   LaserStart_Ext()
   LIN {X -4.398, Y -8.592, Z 58.650}
   LaserEnd_Ext()
   LIN {X -4.398, Y 35.301, Z 58.650}
   LaserStart_Ext()
   LIN {X -4.398, Y 43.362, Z 58.650}
   LaserEnd_Ext()
   LIN {X -5.398, Y 42.761, Z 58.650}
   LaserStart_Ext()
   LIN {X -5.398, Y 38.302, Z 58.650}
   LaserEnd_Ext()
   LIN {X -5.398, Y -11.620, Z 58.650}
   LaserStart_Ext()
   LIN {X -5.398, Y -17.297, Z 58.650}
   LaserEnd_Ext()
   LIN {X -5.398, Y -23.853, Z 58.650}
   LaserStart_Ext()
   LIN {X -5.398, Y -26.825, Z 58.650}
   LaserEnd_Ext()
   LIN {X -6.398, Y -25.920, Z 58.650}
   LaserStart_Ext()
   LIN {X -6.398, Y -20.860, Z 58.650}
   LaserEnd_Ext()
   LIN {X -6.398, Y -20.280, Z 58.650}
   LaserStart_Ext()
   LIN {X -6.398, Y -14.254, Z 58.650}
   LaserEnd_Ext()
   LIN {X -7.398, Y -16.609, Z 58.650}
   LaserStart_Ext()
   LIN {X -7.398, Y -24.292, Z 58.650}
   LaserEnd_Ext()
   LIN {X -8.398, Y -20.132, Z 58.650}
   LaserStart_Ext()
   LIN {X -8.398, Y -20.032, Z 58.650}
   LaserEnd_Ext()
   LIN {X 3.651, Y -23.553, Z 59.500}
   LaserStart_Ext()
   LIN {X 2.587, Y -24.503, Z 59.500} C_DIS
   LIN {X 2.113, Y -24.924, Z 59.500} C_DIS
   LIN {X 1.058, Y -25.251, Z 59.500} C_DIS
   LIN {X 0.034, Y -25.570, Z 59.500} C_DIS
   LIN {X -0.602, Y -25.496, Z 59.500} C_DIS
   LIN {X -1.998, Y -25.328, Z 59.500} C_DIS
   LIN {X -3.608, Y -24.363, Z 59.500} C_DIS
   LIN {X -3.770, Y -24.267, Z 59.500} C_DIS
   LIN {X -3.863, Y -24.136, Z 59.500} C_DIS
   LIN {X -4.971, Y -22.565, Z 59.500} C_DIS
   LIN {X -5.320, Y -20.722, Z 59.500} C_DIS
   LIN {X -5.360, Y -20.515, Z 59.500} C_DIS
   LIN {X -4.561, Y -18.080, Z 59.500} C_DIS
   LIN {X -4.452, Y -17.736, Z 59.500} C_DIS
   LIN {X -3.971, Y -17.280, Z 59.500} C_DIS
   LIN {X -2.945, Y -16.315, Z 59.500} C_DIS
   LIN {X -1.929, Y -15.973, Z 59.500} C_DIS
   LIN {X -0.833, Y -15.606, Z 59.500} C_DIS
   LIN {X 0.602, Y -15.764, Z 59.500} C_DIS
   LIN {X 1.276, Y -15.837, Z 59.500} C_DIS
   LIN {X 1.727, Y -16.111, Z 59.500} C_DIS
   LIN {X 3.095, Y -16.936, Z 59.500} C_DIS
   LIN {X 4.204, Y -18.721, Z 59.500} C_DIS
   LIN {X 4.436, Y -19.097, Z 59.500} C_DIS
   LIN {X 4.464, Y -19.505, Z 59.500} C_DIS
   LIN {X 4.594, Y -21.301, Z 59.500} C_DIS
   LIN {X 4.218, Y -22.204, Z 59.500} C_DIS
   LIN {X 3.651, Y -23.553, Z 59.500}
   LaserEnd_Ext()
   LIN {X 4.394, Y 32.266, Z 59.500}
   LaserStart_Ext()
   LIN {X 4.205, Y 32.926, Z 59.500} C_DIS
   LIN {X 4.104, Y 33.232, Z 59.500} C_DIS
   LIN {X 3.655, Y 34.459, Z 59.500} C_DIS
   LIN {X 2.800, Y 36.803, Z 59.500} C_DIS
   LIN {X 2.432, Y 37.727, Z 59.500} C_DIS
   LIN {X 1.920, Y 39.018, Z 59.500} C_DIS
   LIN {X 1.377, Y 40.311, Z 59.500} C_DIS
   LIN {X 1.096, Y 40.976, Z 59.500} C_DIS
   LIN {X 0.783, Y 41.682, Z 59.500} C_DIS
   LIN {X 0.407, Y 42.537, Z 59.500} C_DIS
   LIN {X 0.002, Y 43.122, Z 59.500} C_DIS
   LIN {X -0.432, Y 43.746, Z 59.500} C_DIS
   LIN {X -1.529, Y 44.437, Z 59.500} C_DIS
   LIN {X -1.904, Y 44.674, Z 59.500} C_DIS
   LIN {X -2.162, Y 44.707, Z 59.500} C_DIS
   LIN {X -3.636, Y 44.890, Z 59.500} C_DIS
   LIN {X -5.139, Y 44.206, Z 59.500} C_DIS
   LIN {X -5.994, Y 43.806, Z 59.500} C_DIS
   LIN {X -6.906, Y 42.487, Z 59.500} C_DIS
   LIN {X -7.065, Y 41.690, Z 59.500} C_DIS
   LIN {X -7.219, Y 40.882, Z 59.500} C_DIS
   LIN {X -7.097, Y 40.290, Z 59.500} C_DIS
   LIN {X -6.944, Y 39.491, Z 59.500} C_DIS
   LIN {X -6.557, Y 38.443, Z 59.500} C_DIS
   LIN {X -6.510, Y 38.317, Z 59.500} C_DIS
   LIN {X -6.469, Y 38.202, Z 59.500} C_DIS
   LIN {X -5.976, Y 36.809, Z 59.500} C_DIS
   LIN {X -5.262, Y 34.603, Z 59.500} C_DIS
   LIN {X -5.221, Y 34.465, Z 59.500} C_DIS
   LIN {X -4.434, Y 31.691, Z 59.500} C_DIS
   LIN {X -4.225, Y 30.834, Z 59.500} C_DIS
   LIN {X -3.738, Y 28.801, Z 59.500} C_DIS
   LIN {X -2.893, Y 24.053, Z 59.500} C_DIS
   LIN {X -2.741, Y 23.217, Z 59.500} C_DIS
   LIN {X -2.690, Y 22.404, Z 59.500} C_DIS
   LIN {X -2.050, Y 13.702, Z 59.500} C_DIS
   LIN {X -2.396, Y 6.398, Z 59.500} C_DIS
   LIN {X -2.420, Y 5.803, Z 59.500} C_DIS
   LIN {X -2.492, Y 5.299, Z 59.500} C_DIS
   LIN {X -3.366, Y -0.609, Z 59.500} C_DIS
   LIN {X -4.427, Y -5.060, Z 59.500} C_DIS
   LIN {X -4.887, Y -6.944, Z 59.500} C_DIS
   LIN {X -5.301, Y -8.237, Z 59.500} C_DIS
   LIN {X -6.048, Y -10.610, Z 59.500} C_DIS
   LIN {X -6.839, Y -12.728, Z 59.500} C_DIS
   LIN {X -7.391, Y -14.184, Z 59.500} C_DIS
   LIN {X -8.023, Y -15.645, Z 59.500} C_DIS
   LIN {X -8.560, Y -16.902, Z 59.500} C_DIS
   LIN {X -8.871, Y -18.130, Z 59.500} C_DIS
   LIN {X -9.347, Y -19.974, Z 59.500} C_DIS
   LIN {X -9.023, Y -22.429, Z 59.500} C_DIS
   LIN {X -8.856, Y -23.652, Z 59.500} C_DIS
   LIN {X -7.892, Y -25.211, Z 59.500} C_DIS
   LIN {X -6.889, Y -26.844, Z 59.500} C_DIS
   LIN {X -6.353, Y -27.250, Z 59.500} C_DIS
   LIN {X -4.562, Y -28.587, Z 59.500} C_DIS
   LIN {X -4.173, Y -28.761, Z 59.500} C_DIS
   LIN {X -2.604, Y -28.918, Z 59.500} C_DIS
   LIN {X 1.615, Y -29.361, Z 59.500} C_DIS
   LIN {X 2.525, Y -28.992, Z 59.500} C_DIS
   LIN {X 4.880, Y -27.881, Z 59.500} C_DIS
   LIN {X 7.304, Y -25.155, Z 59.500} C_DIS
   LIN {X 7.543, Y -24.875, Z 59.500} C_DIS
   LIN {X 7.671, Y -24.507, Z 59.500} C_DIS
   LIN {X 8.526, Y -22.093, Z 59.500} C_DIS
   LIN {X 8.845, Y -20.129, Z 59.500} C_DIS
   LIN {X 9.042, Y -18.870, Z 59.500} C_DIS
   LIN {X 9.234, Y -17.389, Z 59.500} C_DIS
   LIN {X 9.431, Y -15.935, Z 59.500} C_DIS
   LIN {X 9.570, Y -14.614, Z 59.500} C_DIS
   LIN {X 9.814, Y -12.148, Z 59.500} C_DIS
   LIN {X 10.027, Y -8.821, Z 59.500} C_DIS
   LIN {X 10.110, Y -7.369, Z 59.500} C_DIS
   LIN {X 10.159, Y -2.463, Z 59.500} C_DIS
   LIN {X 10.180, Y -0.855, Z 59.500} C_DIS
   LIN {X 10.169, Y -0.533, Z 59.500} C_DIS
   LIN {X 10.095, Y 1.746, Z 59.500} C_DIS
   LIN {X 9.904, Y 5.040, Z 59.500} C_DIS
   LIN {X 9.462, Y 9.698, Z 59.500} C_DIS
   LIN {X 8.824, Y 13.940, Z 59.500} C_DIS
   LIN {X 7.121, Y 22.903, Z 59.500} C_DIS
   LIN {X 6.371, Y 25.828, Z 59.500} C_DIS
   LIN {X 4.394, Y 32.266, Z 59.500}
   LaserEnd_Ext()
   LIN {X -4.229, Y 43.522, Z 59.500}
   LaserStart_Ext()
   LIN {X -1.952, Y 43.522, Z 59.500}
   LaserEnd_Ext()
   LIN {X -0.798, Y 42.522, Z 59.500}
   LaserStart_Ext()
   LIN {X -5.666, Y 42.522, Z 59.500}
   LaserEnd_Ext()
   LIN {X -6.079, Y 41.522, Z 59.500}
   LaserStart_Ext()
   LIN {X -0.239, Y 41.522, Z 59.500}
   LaserEnd_Ext()
   LIN {X 0.202, Y 40.522, Z 59.500}
   LaserStart_Ext()
   LIN {X -6.124, Y 40.522, Z 59.500}
   LaserEnd_Ext()
   LIN {X -5.889, Y 39.522, Z 59.500}
   LaserStart_Ext()
   LIN {X 0.624, Y 39.522, Z 59.500}
   LaserEnd_Ext()
   LIN {X 1.041, Y 38.522, Z 59.500}
   LaserStart_Ext()
   LIN {X -5.522, Y 38.522, Z 59.500}
   LaserEnd_Ext()
   LIN {X -5.168, Y 37.522, Z 59.500}
   LaserStart_Ext()
   LIN {X 1.438, Y 37.522, Z 59.500}
   LaserEnd_Ext()
   LIN {X 1.835, Y 36.522, Z 59.500}
   LaserStart_Ext()
   LIN {X -4.832, Y 36.522, Z 59.500}
   LaserEnd_Ext()
   LIN {X -4.509, Y 35.522, Z 59.500}
   LaserStart_Ext()
   LIN {X 2.203, Y 35.522, Z 59.500}
   LaserEnd_Ext()
   LIN {X 2.568, Y 34.522, Z 59.500}
   LaserStart_Ext()
   LIN {X -4.198, Y 34.522, Z 59.500}
   LaserEnd_Ext()
   LIN {X -3.914, Y 33.522, Z 59.500}
   LaserStart_Ext()
   LIN {X 2.933, Y 33.522, Z 59.500}
   LaserEnd_Ext()
   LIN {X 3.281, Y 32.522, Z 59.500}
   LaserStart_Ext()
   LIN {X -3.630, Y 32.522, Z 59.500}
   LaserEnd_Ext()
   LIN {X -3.363, Y 31.522, Z 59.500}
   LaserStart_Ext()
   LIN {X 3.576, Y 31.522, Z 59.500}
   LaserEnd_Ext()
   LIN {X 3.883, Y 30.522, Z 59.500}
   LaserStart_Ext()
   LIN {X -3.122, Y 30.522, Z 59.500}
   LaserEnd_Ext()
   LIN {X -2.882, Y 29.522, Z 59.500}
   LaserStart_Ext()
   LIN {X 4.190, Y 29.522, Z 59.500}
   LaserEnd_Ext()
   LIN {X 4.498, Y 28.522, Z 59.500}
   LaserStart_Ext()
   LIN {X -2.672, Y 28.522, Z 59.500}
   LaserEnd_Ext()
   LIN {X -2.494, Y 27.522, Z 59.500}
   LaserStart_Ext()
   LIN {X 4.805, Y 27.522, Z 59.500}
   LaserEnd_Ext()
   LIN {X 5.112, Y 26.522, Z 59.500}
   LaserStart_Ext()
   LIN {X -2.316, Y 26.522, Z 59.500}
   LaserEnd_Ext()
   LIN {X -2.138, Y 25.522, Z 59.500}
   LaserStart_Ext()
   LIN {X 5.417, Y 25.522, Z 59.500}
   LaserEnd_Ext()
   LIN {X 5.673, Y 24.522, Z 59.500}
   LaserStart_Ext()
   LIN {X -1.960, Y 24.522, Z 59.500}
   LaserEnd_Ext()
   LIN {X -1.780, Y 23.522, Z 59.500}
   LaserStart_Ext()
   LIN {X 5.930, Y 23.522, Z 59.500}
   LaserEnd_Ext()
   LIN {X 6.175, Y 22.522, Z 59.500}
   LaserStart_Ext()
   LIN {X -1.695, Y 22.522, Z 59.500}
   LaserEnd_Ext()
   LIN {X -1.622, Y 21.522, Z 59.500}
   LaserStart_Ext()
   LIN {X 6.365, Y 21.522, Z 59.500}
   LaserEnd_Ext()
   LIN {X 6.555, Y 20.522, Z 59.500}
   LaserStart_Ext()
   LIN {X -1.549, Y 20.522, Z 59.500}
   LaserEnd_Ext()
   LIN {X -1.475, Y 19.522, Z 59.500}
   LaserStart_Ext()
   LIN {X 6.745, Y 19.522, Z 59.500}
   LaserEnd_Ext()
   LIN {X 6.936, Y 18.522, Z 59.500}
   LaserStart_Ext()
   LIN {X -1.401, Y 18.522, Z 59.500}
   LaserEnd_Ext()
   LIN {X -1.328, Y 17.522, Z 59.500}
   LaserStart_Ext()
   LIN {X 7.126, Y 17.522, Z 59.500}
   LaserEnd_Ext()
   LIN {X 7.316, Y 16.522, Z 59.500}
   LaserStart_Ext()
   LIN {X -1.254, Y 16.522, Z 59.500}
   LaserEnd_Ext()
   LIN {X -1.181, Y 15.522, Z 59.500}
   LaserStart_Ext()
   LIN {X 7.506, Y 15.522, Z 59.500}
   LaserEnd_Ext()
   LIN {X 7.696, Y 14.522, Z 59.500}
   LaserStart_Ext()
   LIN {X -1.107, Y 14.522, Z 59.500}
   LaserEnd_Ext()
   LIN {X -1.057, Y 13.522, Z 59.500}
   LaserStart_Ext()
   LIN {X 7.876, Y 13.522, Z 59.500}
   LaserEnd_Ext()
   LIN {X 8.027, Y 12.522, Z 59.500}
   LaserStart_Ext()
   LIN {X -1.105, Y 12.522, Z 59.500}
   LaserEnd_Ext()
   LIN {X -1.152, Y 11.522, Z 59.500}
   LaserStart_Ext()
   LIN {X 8.177, Y 11.522, Z 59.500}
   LaserEnd_Ext()
   LIN {X 8.327, Y 10.522, Z 59.500}
   LaserStart_Ext()
   LIN {X -1.199, Y 10.522, Z 59.500}
   LaserEnd_Ext()
   LIN {X -1.247, Y 9.522, Z 59.500}
   LaserStart_Ext()
   LIN {X 8.475, Y 9.522, Z 59.500}
   LaserEnd_Ext()
   LIN {X 8.569, Y 8.522, Z 59.500}
   LaserStart_Ext()
   LIN {X -1.294, Y 8.522, Z 59.500}
   LaserEnd_Ext()
   LIN {X -1.341, Y 7.522, Z 59.500}
   LaserStart_Ext()
   LIN {X 8.664, Y 7.522, Z 59.500}
   LaserEnd_Ext()
   LIN {X 8.759, Y 6.522, Z 59.500}
   LaserStart_Ext()
   LIN {X -1.389, Y 6.522, Z 59.500}
   LaserEnd_Ext()
   LIN {X -1.450, Y 5.522, Z 59.500}
   LaserStart_Ext()
   LIN {X 8.853, Y 5.522, Z 59.500}
   LaserEnd_Ext()
   LIN {X 8.932, Y 4.522, Z 59.500}
   LaserStart_Ext()
   LIN {X -1.596, Y 4.522, Z 59.500}
   LaserEnd_Ext()
   LIN {X -1.744, Y 3.522, Z 59.500}
   LaserStart_Ext()
   LIN {X 8.990, Y 3.522, Z 59.500}
   LaserEnd_Ext()
   LIN {X 9.049, Y 2.522, Z 59.500}
   LaserStart_Ext()
   LIN {X -1.892, Y 2.522, Z 59.500}
   LaserEnd_Ext()
   LIN {X -2.040, Y 1.522, Z 59.500}
   LaserStart_Ext()
   LIN {X 9.102, Y 1.522, Z 59.500}
   LaserEnd_Ext()
   LIN {X 9.135, Y 0.522, Z 59.500}
   LaserStart_Ext()
   LIN {X -2.188, Y 0.522, Z 59.500}
   LaserEnd_Ext()
   LIN {X -2.336, Y -0.478, Z 59.500}
   LaserStart_Ext()
   LIN {X 9.167, Y -0.478, Z 59.500}
   LaserEnd_Ext()
   LIN {X 9.172, Y -1.478, Z 59.500}
   LaserStart_Ext()
   LIN {X -2.545, Y -1.478, Z 59.500}
   LaserEnd_Ext()
   LIN {X -2.784, Y -2.478, Z 59.500}
   LaserStart_Ext()
   LIN {X 9.159, Y -2.478, Z 59.500}
   LaserEnd_Ext()
   LIN {X 9.149, Y -3.478, Z 59.500}
   LaserStart_Ext()
   LIN {X -3.022, Y -3.478, Z 59.500}
   LaserEnd_Ext()
   LIN {X -3.260, Y -4.478, Z 59.500}
   LaserStart_Ext()
   LIN {X 9.139, Y -4.478, Z 59.500}
   LaserEnd_Ext()
   LIN {X 9.129, Y -5.478, Z 59.500}
   LaserStart_Ext()
   LIN {X -3.500, Y -5.478, Z 59.500}
   LaserEnd_Ext()
   LIN {X -3.744, Y -6.478, Z 59.500}
   LaserStart_Ext()
   LIN {X 9.119, Y -6.478, Z 59.500}
   LaserEnd_Ext()
   LIN {X 9.102, Y -7.478, Z 59.500}
   LaserStart_Ext()
   LIN {X -4.008, Y -7.478, Z 59.500}
   LaserEnd_Ext()
   LIN {X -4.329, Y -8.478, Z 59.500}
   LaserStart_Ext()
   LIN {X 9.045, Y -8.478, Z 59.500}
   LaserEnd_Ext()
   LIN {X 8.983, Y -9.478, Z 59.500}
   LaserStart_Ext()
   LIN {X -4.644, Y -9.478, Z 59.500}
   LaserEnd_Ext()
   LIN {X -4.958, Y -10.478, Z 59.500}
   LaserStart_Ext()
   LIN {X 8.919, Y -10.478, Z 59.500}
   LaserEnd_Ext()
   LIN {X 8.855, Y -11.478, Z 59.500}
   LaserStart_Ext()
   LIN {X -5.305, Y -11.478, Z 59.500}
   LaserEnd_Ext()
   LIN {X -5.678, Y -12.478, Z 59.500}
   LaserStart_Ext()
   LIN {X 8.776, Y -12.478, Z 59.500}
   LaserEnd_Ext()
   LIN {X 8.677, Y -13.478, Z 59.500}
   LaserStart_Ext()
   LIN {X -6.054, Y -13.478, Z 59.500}
   LaserEnd_Ext()
   LIN {X -6.434, Y -14.478, Z 59.500}
   LaserStart_Ext()
   LIN {X 8.579, Y -14.478, Z 59.500}
   LaserEnd_Ext()
   LIN {X 8.473, Y -15.478, Z 59.500}
   LaserStart_Ext()
   LIN {X 2.614, Y -15.478, Z 59.500}
   LaserEnd_Ext()
   LIN {X -3.490, Y -15.478, Z 59.500}
   LaserStart_Ext()
   LIN {X -6.862, Y -15.478, Z 59.500}
   LaserEnd_Ext()
   LIN {X -7.292, Y -16.478, Z 59.500}
   LaserStart_Ext()
   LIN {X -4.578, Y -16.478, Z 59.500}
   LaserEnd_Ext()
   LIN {X 3.988, Y -16.478, Z 59.500}
   LaserStart_Ext()
   LIN {X 8.348, Y -16.478, Z 59.500}
   LaserEnd_Ext()
   LIN {X 8.214, Y -17.478, Z 59.500}
   LaserStart_Ext()
   LIN {X 4.609, Y -17.478, Z 59.500}
   LaserEnd_Ext()
   LIN {X -5.419, Y -17.478, Z 59.500}
   LaserStart_Ext()
   LIN {X -7.675, Y -17.478, Z 59.500}
   LaserEnd_Ext()
   LIN {X -7.928, Y -18.478, Z 59.500}
   LaserStart_Ext()
   LIN {X -5.744, Y -18.478, Z 59.500}
   LaserEnd_Ext()
   LIN {X 5.229, Y -18.478, Z 59.500}
   LaserStart_Ext()
   LIN {X 8.085, Y -18.478, Z 59.500}
   LaserEnd_Ext()
   LIN {X 7.935, Y -19.478, Z 59.500}
   LaserStart_Ext()
   LIN {X 5.464, Y -19.478, Z 59.500}
   LaserEnd_Ext()
   LIN {X -6.072, Y -19.478, Z 59.500}
   LaserStart_Ext()
   LIN {X -8.186, Y -19.478, Z 59.500}
   LaserEnd_Ext()
   LIN {X -8.272, Y -20.478, Z 59.500}
   LaserStart_Ext()
   LIN {X -6.358, Y -20.478, Z 59.500}
   LaserEnd_Ext()
   LIN {X 5.537, Y -20.478, Z 59.500}
   LaserStart_Ext()
   LIN {X 7.775, Y -20.478, Z 59.500}
   LaserEnd_Ext()
   LIN {X 7.612, Y -21.478, Z 59.500}
   LaserStart_Ext()
   LIN {X 5.577, Y -21.478, Z 59.500}
   LaserEnd_Ext()
   LIN {X -6.194, Y -21.478, Z 59.500}
   LaserStart_Ext()
   LIN {X -8.140, Y -21.478, Z 59.500}
   LaserEnd_Ext()
   LIN {X -8.007, Y -22.478, Z 59.500}
   LaserStart_Ext()
   LIN {X -6.005, Y -22.478, Z 59.500}
   LaserEnd_Ext()
   LIN {X 5.187, Y -22.478, Z 59.500}
   LaserStart_Ext()
   LIN {X 7.328, Y -22.478, Z 59.500}
   LaserEnd_Ext()
   LIN {X 6.974, Y -23.478, Z 59.500}
   LaserStart_Ext()
   LIN {X 4.768, Y -23.478, Z 59.500}
   LaserEnd_Ext()
   LIN {X -5.550, Y -23.478, Z 59.500}
   LaserStart_Ext()
   LIN {X -7.787, Y -23.478, Z 59.500}
   LaserEnd_Ext()
   LIN {X -7.169, Y -24.478, Z 59.500}
   LaserStart_Ext()
   LIN {X -4.845, Y -24.478, Z 59.500}
   LaserEnd_Ext()
   LIN {X 4.117, Y -24.478, Z 59.500}
   LaserStart_Ext()
   LIN {X 6.567, Y -24.478, Z 59.500}
   LaserEnd_Ext()
   LIN {X 5.678, Y -25.478, Z 59.500}
   LaserStart_Ext()
   LIN {X 2.995, Y -25.478, Z 59.500}
   LaserEnd_Ext()
   LIN {X -3.692, Y -25.478, Z 59.500}
   LaserStart_Ext()
   LIN {X -6.554, Y -25.478, Z 59.500}
   LaserEnd_Ext()
   LIN {X -5.715, Y -26.478, Z 59.500}
   LaserStart_Ext()
   LIN {X -0.805, Y -26.478, Z 59.500}
   LaserEnd_Ext()
   LIN {X 0.480, Y -26.478, Z 59.500}
   LaserStart_Ext()
   LIN {X 4.789, Y -26.478, Z 59.500}
   LaserEnd_Ext()
   LIN {X 3.390, Y -27.478, Z 59.500}
   LaserStart_Ext()
   LIN {X -4.375, Y -27.478, Z 59.500}
   LaserEnd_Ext()
   LIN {X 4.510, Y -19.033, Z 60.350}
   LaserStart_Ext()
   LIN {X 4.595, Y -20.145, Z 60.350} C_DIS
   LIN {X 4.674, Y -21.238, Z 60.350} C_DIS
   LIN {X 3.955, Y -22.965, Z 60.350} C_DIS
   LIN {X 3.731, Y -23.500, Z 60.350} C_DIS
   LIN {X 2.852, Y -24.285, Z 60.350} C_DIS
   LIN {X 2.203, Y -24.865, Z 60.350} C_DIS
   LIN {X 1.605, Y -25.055, Z 60.350} C_DIS
   LIN {X 0.124, Y -25.517, Z 60.350} C_DIS
   LIN {X -1.796, Y -25.293, Z 60.350} C_DIS
   LIN {X -1.908, Y -25.280, Z 60.350} C_DIS
   LIN {X -2.037, Y -25.202, Z 60.350} C_DIS
   LIN {X -3.683, Y -24.223, Z 60.350} C_DIS
   LIN {X -4.626, Y -22.895, Z 60.350} C_DIS
   LIN {X -4.888, Y -22.524, Z 60.350} C_DIS
   LIN {X -4.971, Y -22.087, Z 60.350} C_DIS
   LIN {X -5.282, Y -20.474, Z 60.350} C_DIS
   LIN {X -4.779, Y -18.944, Z 60.350} C_DIS
   LIN {X -4.385, Y -17.701, Z 60.350} C_DIS
   LIN {X -3.046, Y -16.431, Z 60.350} C_DIS
   LIN {X -2.872, Y -16.266, Z 60.350} C_DIS
   LIN {X -2.533, Y -16.155, Z 60.350} C_DIS
   LIN {X -0.726, Y -15.551, Z 60.350} C_DIS
   LIN {X 0.562, Y -15.693, Z 60.350} C_DIS
   LIN {X 1.343, Y -15.781, Z 60.350} C_DIS
   LIN {X 2.224, Y -16.309, Z 60.350} C_DIS
   LIN {X 3.164, Y -16.876, Z 60.350} C_DIS
   LIN {X 3.788, Y -17.879, Z 60.350} C_DIS
   LIN {X 4.510, Y -19.033, Z 60.350}
   LaserEnd_Ext()
   LIN {X -2.258, Y 9.479, Z 60.350}
   LaserStart_Ext()
   LIN {X -2.407, Y 5.813, Z 60.350} C_DIS
   LIN {X -2.852, Y 2.701, Z 60.350} C_DIS
   LIN {X -3.336, Y -0.567, Z 60.350} C_DIS
   LIN {X -4.593, Y -5.843, Z 60.350} C_DIS
   LIN {X -4.841, Y -6.902, Z 60.350} C_DIS
   LIN {X -4.992, Y -7.389, Z 60.350} C_DIS
   LIN {X -5.991, Y -10.566, Z 60.350} C_DIS
   LIN {X -7.288, Y -14.040, Z 60.350} C_DIS
   LIN {X -7.326, Y -14.143, Z 60.350} C_DIS
   LIN {X -8.491, Y -16.870, Z 60.350} C_DIS
   LIN {X -9.183, Y -19.603, Z 60.350} C_DIS
   LIN {X -9.270, Y -19.943, Z 60.350} C_DIS
   LIN {X -9.211, Y -20.396, Z 60.350} C_DIS
   LIN {X -8.770, Y -23.620, Z 60.350} C_DIS
   LIN {X -7.071, Y -26.369, Z 60.350} C_DIS
   LIN {X -6.796, Y -26.807, Z 60.350} C_DIS
   LIN {X -6.119, Y -27.310, Z 60.350} C_DIS
   LIN {X -4.465, Y -28.545, Z 60.350} C_DIS
   LIN {X -4.282, Y -28.626, Z 60.350} C_DIS
   LIN {X -3.546, Y -28.700, Z 60.350} C_DIS
   LIN {X 0.598, Y -29.136, Z 60.350} C_DIS
   LIN {X 1.661, Y -29.303, Z 60.350} C_DIS
   LIN {X 1.885, Y -29.267, Z 60.350} C_DIS
   LIN {X 2.307, Y -29.056, Z 60.350} C_DIS
   LIN {X 5.052, Y -27.762, Z 60.350} C_DIS
   LIN {X 6.445, Y -26.195, Z 60.350} C_DIS
   LIN {X 7.632, Y -24.802, Z 60.350} C_DIS
   LIN {X 8.273, Y -22.964, Z 60.350} C_DIS
   LIN {X 8.608, Y -22.020, Z 60.350} C_DIS
   LIN {X 8.733, Y -21.251, Z 60.350} C_DIS
   LIN {X 9.117, Y -18.796, Z 60.350} C_DIS
   LIN {X 9.492, Y -15.906, Z 60.350} C_DIS
   LIN {X 9.872, Y -12.072, Z 60.350} C_DIS
   LIN {X 9.980, Y -10.384, Z 60.350} C_DIS
   LIN {X 10.157, Y -7.292, Z 60.350} C_DIS
   LIN {X 10.207, Y -2.359, Z 60.350} C_DIS
   LIN {X 10.212, Y -0.778, Z 60.350} C_DIS
   LIN {X 10.147, Y 1.211, Z 60.350} C_DIS
   LIN {X 9.913, Y 5.225, Z 60.350} C_DIS
   LIN {X 9.551, Y 9.056, Z 60.350} C_DIS
   LIN {X 8.711, Y 14.640, Z 60.350} C_DIS
   LIN {X 7.244, Y 22.355, Z 60.350} C_DIS
   LIN {X 6.267, Y 26.166, Z 60.350} C_DIS
   LIN {X 4.588, Y 31.635, Z 60.350} C_DIS
   LIN {X 4.129, Y 33.085, Z 60.350} C_DIS
   LIN {X 3.831, Y 33.896, Z 60.350} C_DIS
   LIN {X 2.825, Y 36.652, Z 60.350} C_DIS
   LIN {X 1.935, Y 38.888, Z 60.350} C_DIS
   LIN {X 1.013, Y 41.069, Z 60.350} C_DIS
   LIN {X 0.610, Y 41.980, Z 60.350} C_DIS
   LIN {X 0.337, Y 42.590, Z 60.350} C_DIS
   LIN {X -0.125, Y 43.253, Z 60.350} C_DIS
   LIN {X -0.504, Y 43.798, Z 60.350} C_DIS
   LIN {X -0.985, Y 44.101, Z 60.350} C_DIS
   LIN {X -1.978, Y 44.722, Z 60.350} C_DIS
   LIN {X -3.602, Y 44.920, Z 60.350} C_DIS
   LIN {X -3.711, Y 44.934, Z 60.350} C_DIS
   LIN {X -6.089, Y 43.823, Z 60.350} C_DIS
   LIN {X -6.809, Y 42.780, Z 60.350} C_DIS
   LIN {X -7.001, Y 42.451, Z 60.350} C_DIS
   LIN {X -7.125, Y 41.669, Z 60.350} C_DIS
   LIN {X -7.284, Y 40.842, Z 60.350} C_DIS
   LIN {X -7.128, Y 40.090, Z 60.350} C_DIS
   LIN {X -7.006, Y 39.527, Z 60.350} C_DIS
   LIN {X -6.865, Y 39.149, Z 60.350} C_DIS
   LIN {X -6.570, Y 38.354, Z 60.350} C_DIS
   LIN {X -6.069, Y 36.948, Z 60.350} C_DIS
   LIN {X -6.033, Y 36.848, Z 60.350} C_DIS
   LIN {X -5.297, Y 34.594, Z 60.350} C_DIS
   LIN {X -4.642, Y 32.293, Z 60.350} C_DIS
   LIN {X -4.417, Y 31.500, Z 60.350} C_DIS
   LIN {X -4.360, Y 31.267, Z 60.350} C_DIS
   LIN {X -3.726, Y 28.619, Z 60.350} C_DIS
   LIN {X -2.933, Y 24.163, Z 60.350} C_DIS
   LIN {X -2.761, Y 23.224, Z 60.350} C_DIS
   LIN {X -2.587, Y 21.107, Z 60.350} C_DIS
   LIN {X -2.052, Y 13.832, Z 60.350} C_DIS
   LIN {X -2.258, Y 9.479, Z 60.350}
   LaserEnd_Ext()
   LIN {X -7.280, Y -24.129, Z 60.350}
   LaserStart_Ext()
   LIN {X -7.280, Y -16.581, Z 60.350}
   LaserEnd_Ext()
   LIN {X -6.280, Y -14.199, Z 60.350}
   LaserStart_Ext()
   LIN {X -6.280, Y -20.432, Z 60.350}
   LaserEnd_Ext()
   LIN {X -6.280, Y -20.511, Z 60.350}
   LaserStart_Ext()
   LIN {X -6.280, Y -25.747, Z 60.350}
   LaserEnd_Ext()
   LIN {X -5.280, Y -26.688, Z 60.350}
   LaserStart_Ext()
   LIN {X -5.280, Y -23.701, Z 60.350}
   LaserEnd_Ext()
   LIN {X -5.280, Y -17.257, Z 60.350}
   LaserStart_Ext()
   LIN {X -5.280, Y -11.519, Z 60.350}
   LaserEnd_Ext()
   LIN {X -5.280, Y 37.713, Z 60.350}
   LaserStart_Ext()
   LIN {X -5.280, Y 43.097, Z 60.350}
   LaserEnd_Ext()
   LIN {X -4.280, Y 43.565, Z 60.350}
   LaserStart_Ext()
   LIN {X -4.280, Y 34.672, Z 60.350}
   LaserEnd_Ext()
   LIN {X -4.280, Y -8.458, Z 60.350}
   LaserStart_Ext()
   LIN {X -4.280, Y -16.223, Z 60.350}
   LaserEnd_Ext()
   LIN {X -4.280, Y -25.025, Z 60.350}
   LaserStart_Ext()
   LIN {X -4.280, Y -27.435, Z 60.350}
   LaserEnd_Ext()
   LIN {X -3.280, Y -27.722, Z 60.350}
   LaserStart_Ext()
   LIN {X -3.280, Y -25.626, Z 60.350}
   LaserEnd_Ext()
   LIN {X -3.280, Y -15.354, Z 60.350}
   LaserStart_Ext()
   LIN {X -3.280, Y -4.648, Z 60.350}
   LaserEnd_Ext()
   LIN {X -3.280, Y 31.049, Z 60.350}
   LaserStart_Ext()
   LIN {X -3.280, Y 43.874, Z 60.350}
   LaserEnd_Ext()
   LIN {X -2.280, Y 43.731, Z 60.350}
   LaserStart_Ext()
   LIN {X -2.280, Y 26.199, Z 60.350}
   LaserEnd_Ext()
   LIN {X -2.280, Y -0.264, Z 60.350}
   LaserStart_Ext()
   LIN {X -2.280, Y -15.017, Z 60.350}
   LaserEnd_Ext()
   LIN {X -2.280, Y -26.206, Z 60.350}
   LaserStart_Ext()
   LIN {X -2.280, Y -27.828, Z 60.350}
   LaserEnd_Ext()
   LIN {X -1.280, Y -27.933, Z 60.350}
   LaserStart_Ext()
   LIN {X -1.280, Y -26.360, Z 60.350}
   LaserEnd_Ext()
   LIN {X -1.280, Y -14.682, Z 60.350}
   LaserStart_Ext()
   LIN {X -1.280, Y 8.916, Z 60.350}
   LaserEnd_Ext()
   LIN {X -1.280, Y 16.973, Z 60.350}
   LaserStart_Ext()
   LIN {X -1.280, Y 43.104, Z 60.350}
   LaserEnd_Ext()
   LIN {X -0.280, Y 41.519, Z 60.350}
   LaserStart_Ext()
   LIN {X -0.280, Y -14.595, Z 60.350}
   LaserEnd_Ext()
   LIN {X -0.280, Y -26.476, Z 60.350}
   LaserStart_Ext()
   LIN {X -0.280, Y -28.038, Z 60.350}
   LaserEnd_Ext()
   LIN {X 0.720, Y -28.144, Z 60.350}
   LaserStart_Ext()
   LIN {X 0.720, Y -26.378, Z 60.350}
   LaserEnd_Ext()
   LIN {X 0.720, Y -14.705, Z 60.350}
   LaserStart_Ext()
   LIN {X 0.720, Y 39.193, Z 60.350}
   LaserEnd_Ext()
   LIN {X 1.720, Y 36.723, Z 60.350}
   LaserStart_Ext()
   LIN {X 1.720, Y -14.857, Z 60.350}
   LaserEnd_Ext()
   LIN {X 1.720, Y -26.066, Z 60.350}
   LaserStart_Ext()
   LIN {X 1.720, Y -28.231, Z 60.350}
   LaserEnd_Ext()
   LIN {X 2.720, Y -27.756, Z 60.350}
   LaserStart_Ext()
   LIN {X 2.720, Y -25.720, Z 60.350}
   LaserEnd_Ext()
   LIN {X 2.720, Y -15.440, Z 60.350}
   LaserStart_Ext()
   LIN {X 2.720, Y 34.022, Z 60.350}
   LaserEnd_Ext()
   LIN {X 3.720, Y 31.054, Z 60.350}
   LaserStart_Ext()
   LIN {X 3.720, Y -16.046, Z 60.350}
   LaserEnd_Ext()
   LIN {X 3.720, Y -24.850, Z 60.350}
   LaserStart_Ext()
   LIN {X 3.720, Y -27.284, Z 60.350}
   LaserEnd_Ext()
   LIN {X 4.720, Y -26.630, Z 60.350}
   LaserStart_Ext()
   LIN {X 4.720, Y -23.726, Z 60.350}
   LaserEnd_Ext()
   LIN {X 4.720, Y -17.484, Z 60.350}
   LaserStart_Ext()
   LIN {X 4.720, Y 27.798, Z 60.350}
   LaserEnd_Ext()
   LIN {X 5.720, Y 24.274, Z 60.350}
   LaserStart_Ext()
   LIN {X 5.720, Y -25.504, Z 60.350}
   LaserEnd_Ext()
   LIN {X 6.720, Y -24.331, Z 60.350}
   LaserStart_Ext()
   LIN {X 6.720, Y 19.757, Z 60.350}
   LaserEnd_Ext()
   LIN {X 7.720, Y 14.497, Z 60.350}
   LaserStart_Ext()
   LIN {X 7.720, Y -21.247, Z 60.350}
   LaserEnd_Ext()
   LIN {X 8.720, Y -13.563, Z 60.350}
   LaserStart_Ext()
   LIN {X 8.720, Y 7.218, Z 60.350}
   LaserEnd_Ext()
   LIN {X -4.805, Y -22.482, Z 61.200}
   LaserStart_Ext()
   LIN {X -5.006, Y -21.460, Z 61.200} C_DIS
   LIN {X -5.204, Y -20.434, Z 61.200} C_DIS
   LIN {X -4.998, Y -19.808, Z 61.200} C_DIS
   LIN {X -4.319, Y -17.665, Z 61.200} C_DIS
   LIN {X -3.894, Y -17.263, Z 61.200} C_DIS
   LIN {X -2.768, Y -16.199, Z 61.200} C_DIS
   LIN {X -0.652, Y -15.507, Z 61.200} C_DIS
   LIN {X 1.410, Y -15.725, Z 61.200} C_DIS
   LIN {X 2.830, Y -16.576, Z 61.200} C_DIS
   LIN {X 3.234, Y -16.815, Z 61.200} C_DIS
   LIN {X 3.564, Y -17.339, Z 61.200} C_DIS
   LIN {X 4.585, Y -18.970, Z 61.200} C_DIS
   LIN {X 4.720, Y -20.745, Z 61.200} C_DIS
   LIN {X 4.754, Y -21.174, Z 61.200} C_DIS
   LIN {X 4.663, Y -21.393, Z 61.200} C_DIS
   LIN {X 3.810, Y -23.447, Z 61.200} C_DIS
   LIN {X 3.493, Y -23.733, Z 61.200} C_DIS
   LIN {X 2.295, Y -24.805, Z 61.200} C_DIS
   LIN {X 0.472, Y -25.383, Z 61.200} C_DIS
   LIN {X 0.214, Y -25.464, Z 61.200} C_DIS
   LIN {X -0.167, Y -25.419, Z 61.200} C_DIS
   LIN {X -1.819, Y -25.231, Z 61.200} C_DIS
   LIN {X -2.892, Y -24.598, Z 61.200} C_DIS
   LIN {X -3.596, Y -24.178, Z 61.200} C_DIS
   LIN {X -4.157, Y -23.389, Z 61.200} C_DIS
   LIN {X -4.805, Y -22.482, Z 61.200}
   LaserEnd_Ext()
   LIN {X -4.066, Y 29.904, Z 61.200}
   LaserStart_Ext()
   LIN {X -3.715, Y 28.437, Z 61.200} C_DIS
   LIN {X -3.402, Y 26.682, Z 61.200} C_DIS
   LIN {X -2.820, Y 23.496, Z 61.200} C_DIS
   LIN {X -2.226, Y 16.304, Z 61.200} C_DIS
   LIN {X -2.053, Y 13.961, Z 61.200} C_DIS
   LIN {X -2.120, Y 12.560, Z 61.200} C_DIS
   LIN {X -2.394, Y 5.822, Z 61.200} C_DIS
   LIN {X -3.212, Y 0.104, Z 61.200} C_DIS
   LIN {X -3.305, Y -0.524, Z 61.200} C_DIS
   LIN {X -3.546, Y -1.536, Z 61.200} C_DIS
   LIN {X -4.793, Y -6.855, Z 61.200} C_DIS
   LIN {X -5.550, Y -9.299, Z 61.200} C_DIS
   LIN {X -5.935, Y -10.522, Z 61.200} C_DIS
   LIN {X -6.434, Y -11.859, Z 61.200} C_DIS
   LIN {X -7.263, Y -14.108, Z 61.200} C_DIS
   LIN {X -7.800, Y -15.384, Z 61.200} C_DIS
   LIN {X -8.421, Y -16.837, Z 61.200} C_DIS
   LIN {X -8.894, Y -18.703, Z 61.200} C_DIS
   LIN {X -9.193, Y -19.912, Z 61.200} C_DIS
   LIN {X -8.996, Y -21.313, Z 61.200} C_DIS
   LIN {X -8.685, Y -23.588, Z 61.200} C_DIS
   LIN {X -7.739, Y -25.118, Z 61.200} C_DIS
   LIN {X -6.703, Y -26.770, Z 61.200} C_DIS
   LIN {X -4.467, Y -28.430, Z 61.200} C_DIS
   LIN {X -4.368, Y -28.502, Z 61.200} C_DIS
   LIN {X -4.023, Y -28.583, Z 61.200} C_DIS
   LIN {X 0.904, Y -29.357, Z 61.200} C_DIS
   LIN {X 2.152, Y -29.158, Z 61.200} C_DIS
   LIN {X 4.508, Y -27.980, Z 61.200} C_DIS
   LIN {X 5.223, Y -27.643, Z 61.200} C_DIS
   LIN {X 5.586, Y -27.235, Z 61.200} C_DIS
   LIN {X 7.722, Y -24.729, Z 61.200} C_DIS
   LIN {X 8.558, Y -22.333, Z 61.200} C_DIS
   LIN {X 8.690, Y -21.946, Z 61.200} C_DIS
   LIN {X 8.789, Y -21.290, Z 61.200} C_DIS
   LIN {X 9.191, Y -18.721, Z 61.200} C_DIS
   LIN {X 9.416, Y -16.985, Z 61.200} C_DIS
   LIN {X 9.566, Y -15.784, Z 61.200} C_DIS
   LIN {X 9.920, Y -12.110, Z 61.200} C_DIS
   LIN {X 9.931, Y -11.995, Z 61.200} C_DIS
   LIN {X 10.204, Y -7.215, Z 61.200} C_DIS
   LIN {X 10.232, Y -4.510, Z 61.200} C_DIS
   LIN {X 10.244, Y -0.701, Z 61.200} C_DIS
   LIN {X 10.199, Y 0.676, Z 61.200} C_DIS
   LIN {X 9.923, Y 5.410, Z 61.200} C_DIS
   LIN {X 9.639, Y 8.413, Z 61.200} C_DIS
   LIN {X 8.597, Y 15.340, Z 61.200} C_DIS
   LIN {X 7.368, Y 21.808, Z 61.200} C_DIS
   LIN {X 6.164, Y 26.504, Z 61.200} C_DIS
   LIN {X 5.332, Y 29.212, Z 61.200} C_DIS
   LIN {X 4.133, Y 33.002, Z 61.200} C_DIS
   LIN {X 3.353, Y 35.123, Z 61.200} C_DIS
   LIN {X 2.850, Y 36.501, Z 61.200} C_DIS
   LIN {X 2.403, Y 37.624, Z 61.200} C_DIS
   LIN {X 1.858, Y 38.983, Z 61.200} C_DIS
   LIN {X 1.138, Y 40.678, Z 61.200} C_DIS
   LIN {X 0.931, Y 41.160, Z 61.200} C_DIS
   LIN {X 0.676, Y 41.729, Z 61.200} C_DIS
   LIN {X 0.268, Y 42.644, Z 61.200} C_DIS
   LIN {X -0.107, Y 43.180, Z 61.200} C_DIS
   LIN {X -0.577, Y 43.849, Z 61.200} C_DIS
   LIN {X -1.533, Y 44.444, Z 61.200} C_DIS
   LIN {X -2.053, Y 44.770, Z 61.200} C_DIS
   LIN {X -2.502, Y 44.825, Z 61.200} C_DIS
   LIN {X -3.786, Y 44.977, Z 61.200} C_DIS
   LIN {X -5.008, Y 44.389, Z 61.200} C_DIS
   LIN {X -6.183, Y 43.839, Z 61.200} C_DIS
   LIN {X -6.529, Y 43.339, Z 61.200} C_DIS
   LIN {X -7.147, Y 42.279, Z 61.200} C_DIS
   LIN {X -7.255, Y 41.596, Z 61.200} C_DIS
   LIN {X -7.349, Y 40.871, Z 61.200} C_DIS
   LIN {X -7.194, Y 40.142, Z 61.200} C_DIS
   LIN {X -7.068, Y 39.563, Z 61.200} C_DIS
   LIN {X -6.794, Y 38.829, Z 61.200} C_DIS
   LIN {X -6.630, Y 38.391, Z 61.200} C_DIS
   LIN {X -6.526, Y 38.106, Z 61.200} C_DIS
   LIN {X -6.089, Y 36.886, Z 61.200} C_DIS
   LIN {X -5.484, Y 35.051, Z 61.200} C_DIS
   LIN {X -5.348, Y 34.634, Z 61.200} C_DIS
   LIN {X -5.098, Y 33.755, Z 61.200} C_DIS
   LIN {X -4.438, Y 31.455, Z 61.200} C_DIS
   LIN {X -4.066, Y 29.904, Z 61.200}
   LaserEnd_Ext()
   LIN {X -4.231, Y -27.360, Z 61.200}
   LaserStart_Ext()
   LIN {X 3.512, Y -27.360, Z 61.200}
   LaserEnd_Ext()
   LIN {X 5.018, Y -26.360, Z 61.200}
   LaserStart_Ext()
   LIN {X 0.699, Y -26.360, Z 61.200}
   LaserEnd_Ext()
   LIN {X -0.743, Y -26.360, Z 61.200}
   LaserStart_Ext()
   LIN {X -5.578, Y -26.360, Z 61.200}
   LaserEnd_Ext()
   LIN {X -6.407, Y -25.360, Z 61.200}
   LaserStart_Ext()
   LIN {X -3.566, Y -25.360, Z 61.200}
   LaserEnd_Ext()
   LIN {X 3.174, Y -25.360, Z 61.200}
   LaserStart_Ext()
   LIN {X 5.870, Y -25.360, Z 61.200}
   LaserEnd_Ext()
   LIN {X 6.723, Y -24.360, Z 61.200}
   LaserStart_Ext()
   LIN {X 4.290, Y -24.360, Z 61.200}
   LaserEnd_Ext()
   LIN {X -4.694, Y -24.360, Z 61.200}
   LaserStart_Ext()
   LIN {X -7.032, Y -24.360, Z 61.200}
   LaserEnd_Ext()
   LIN {X -7.650, Y -23.360, Z 61.200}
   LaserStart_Ext()
   LIN {X -5.407, Y -23.360, Z 61.200}
   LaserEnd_Ext()
   LIN {X 4.929, Y -23.360, Z 61.200}
   LaserStart_Ext()
   LIN {X 7.140, Y -23.360, Z 61.200}
   LaserEnd_Ext()
   LIN {X 7.489, Y -22.360, Z 61.200}
   LaserStart_Ext()
   LIN {X 5.345, Y -22.360, Z 61.200}
   LaserEnd_Ext()
   LIN {X -5.848, Y -22.360, Z 61.200}
   LaserStart_Ext()
   LIN {X -7.843, Y -22.360, Z 61.200}
   LaserEnd_Ext()
   LIN {X -7.980, Y -21.360, Z 61.200}
   LaserStart_Ext()
   LIN {X -6.043, Y -21.360, Z 61.200}
   LaserEnd_Ext()
   LIN {X 5.736, Y -21.360, Z 61.200}
   LaserStart_Ext()
   LIN {X 7.767, Y -21.360, Z 61.200}
   LaserEnd_Ext()
   LIN {X 7.923, Y -20.360, Z 61.200}
   LaserStart_Ext()
   LIN {X 5.694, Y -20.360, Z 61.200}
   LaserEnd_Ext()
   LIN {X -6.200, Y -20.360, Z 61.200}
   LaserStart_Ext()
   LIN {X -8.120, Y -20.360, Z 61.200}
   LaserEnd_Ext()
   LIN {X -8.026, Y -19.360, Z 61.200}
   LaserStart_Ext()
   LIN {X -5.905, Y -19.360, Z 61.200}
   LaserEnd_Ext()
   LIN {X 5.618, Y -19.360, Z 61.200}
   LaserStart_Ext()
   LIN {X 8.079, Y -19.360, Z 61.200}
   LaserEnd_Ext()
   LIN {X 8.230, Y -18.360, Z 61.200}
   LaserStart_Ext()
   LIN {X 5.383, Y -18.360, Z 61.200}
   LaserEnd_Ext()
   LIN {X -5.588, Y -18.360, Z 61.200}
   LaserStart_Ext()
   LIN {X -7.775, Y -18.360, Z 61.200}
   LaserEnd_Ext()
   LIN {X -7.522, Y -17.360, Z 61.200}
   LaserStart_Ext()
   LIN {X -5.271, Y -17.360, Z 61.200}
   LaserEnd_Ext()
   LIN {X 4.757, Y -17.360, Z 61.200}
   LaserStart_Ext()
   LIN {X 8.359, Y -17.360, Z 61.200}
   LaserEnd_Ext()
   LIN {X 8.486, Y -16.360, Z 61.200}
   LaserStart_Ext()
   LIN {X 4.129, Y -16.360, Z 61.200}
   LaserEnd_Ext()
   LIN {X -4.395, Y -16.360, Z 61.200}
   LaserStart_Ext()
   LIN {X -7.130, Y -16.360, Z 61.200}
   LaserEnd_Ext()
   LIN {X -6.705, Y -15.360, Z 61.200}
   LaserStart_Ext()
   LIN {X -3.311, Y -15.360, Z 61.200}
   LaserEnd_Ext()
   LIN {X 2.747, Y -15.360, Z 61.200}
   LaserStart_Ext()
   LIN {X 8.602, Y -15.360, Z 61.200}
   LaserEnd_Ext()
   LIN {X 8.698, Y -14.360, Z 61.200}
   LaserStart_Ext()
   LIN {X -6.290, Y -14.360, Z 61.200}
   LaserEnd_Ext()
   LIN {X -5.921, Y -13.360, Z 61.200}
   LaserStart_Ext()
   LIN {X 8.794, Y -13.360, Z 61.200}
   LaserEnd_Ext()
   LIN {X 8.891, Y -12.360, Z 61.200}
   LaserStart_Ext()
   LIN {X -5.553, Y -12.360, Z 61.200}
   LaserEnd_Ext()
   LIN {X -5.180, Y -11.360, Z 61.200}
   LaserStart_Ext()
   LIN {X 8.966, Y -11.360, Z 61.200}
   LaserEnd_Ext()
   LIN {X 9.023, Y -10.360, Z 61.200}
   LaserStart_Ext()
   LIN {X -4.836, Y -10.360, Z 61.200}
   LaserEnd_Ext()
   LIN {X -4.522, Y -9.360, Z 61.200}
   LaserStart_Ext()
   LIN {X 9.080, Y -9.360, Z 61.200}
   LaserEnd_Ext()
   LIN {X 9.137, Y -8.360, Z 61.200}
   LaserStart_Ext()
   LIN {X -4.212, Y -8.360, Z 61.200}
   LaserEnd_Ext()
   LIN {X -3.903, Y -7.360, Z 61.200}
   LaserStart_Ext()
   LIN {X 9.195, Y -7.360, Z 61.200}
   LaserEnd_Ext()
   LIN {X 9.213, Y -6.360, Z 61.200}
   LaserStart_Ext()
   LIN {X -3.650, Y -6.360, Z 61.200}
   LaserEnd_Ext()
   LIN {X -3.415, Y -5.360, Z 61.200}
   LaserStart_Ext()
   LIN {X 9.223, Y -5.360, Z 61.200}
   LaserEnd_Ext()
   LIN {X 9.232, Y -4.360, Z 61.200}
   LaserStart_Ext()
   LIN {X -3.181, Y -4.360, Z 61.200}
   LaserEnd_Ext()
   LIN {X -2.946, Y -3.360, Z 61.200}
   LaserStart_Ext()
   LIN {X 9.235, Y -3.360, Z 61.200}
   LaserEnd_Ext()
   LIN {X 9.238, Y -2.360, Z 61.200}
   LaserStart_Ext()
   LIN {X -2.712, Y -2.360, Z 61.200}
   LaserEnd_Ext()
   LIN {X -2.476, Y -1.360, Z 61.200}
   LaserStart_Ext()
   LIN {X 9.242, Y -1.360, Z 61.200}
   LaserEnd_Ext()
   LIN {X 9.232, Y -0.360, Z 61.200}
   LaserStart_Ext()
   LIN {X -2.269, Y -0.360, Z 61.200}
   LaserEnd_Ext()
   LIN {X -2.125, Y 0.640, Z 61.200}
   LaserStart_Ext()
   LIN {X 9.199, Y 0.640, Z 61.200}
   LaserEnd_Ext()
   LIN {X 9.141, Y 1.640, Z 61.200}
   LaserStart_Ext()
   LIN {X -1.982, Y 1.640, Z 61.200}
   LaserEnd_Ext()
   LIN {X -1.839, Y 2.640, Z 61.200}
   LaserStart_Ext()
   LIN {X 9.083, Y 2.640, Z 61.200}
   LaserEnd_Ext()
   LIN {X 9.025, Y 3.640, Z 61.200}
   LaserStart_Ext()
   LIN {X -1.696, Y 3.640, Z 61.200}
   LaserEnd_Ext()
   LIN {X -1.553, Y 4.640, Z 61.200}
   LaserStart_Ext()
   LIN {X 8.966, Y 4.640, Z 61.200}
   LaserEnd_Ext()
   LIN {X 8.897, Y 5.640, Z 61.200}
   LaserStart_Ext()
   LIN {X -1.410, Y 5.640, Z 61.200}
   LaserEnd_Ext()
   LIN {X -1.360, Y 6.640, Z 61.200}
   LaserStart_Ext()
   LIN {X 8.802, Y 6.640, Z 61.200}
   LaserEnd_Ext()
   LIN {X 8.708, Y 7.640, Z 61.200}
   LaserStart_Ext()
   LIN {X -1.319, Y 7.640, Z 61.200}
   LaserEnd_Ext()
   LIN {X -1.278, Y 8.640, Z 61.200}
   LaserStart_Ext()
   LIN {X 8.593, Y 8.640, Z 61.200}
   LaserEnd_Ext()
   LIN {X 8.443, Y 9.640, Z 61.200}
   LaserStart_Ext()
   LIN {X -1.238, Y 9.640, Z 61.200}
   LaserEnd_Ext()
   LIN {X -1.197, Y 10.640, Z 61.200}
   LaserStart_Ext()
   LIN {X 8.293, Y 10.640, Z 61.200}
   LaserEnd_Ext()
   LIN {X 8.142, Y 11.640, Z 61.200}
   LaserStart_Ext()
   LIN {X -1.156, Y 11.640, Z 61.200}
   LaserEnd_Ext()
   LIN {X -1.115, Y 12.640, Z 61.200}
   LaserStart_Ext()
   LIN {X 7.992, Y 12.640, Z 61.200}
   LaserEnd_Ext()
   LIN {X 7.842, Y 13.640, Z 61.200}
   LaserStart_Ext()
   LIN {X -1.067, Y 13.640, Z 61.200}
   LaserEnd_Ext()
   LIN {X -1.101, Y 14.640, Z 61.200}
   LaserStart_Ext()
   LIN {X 7.691, Y 14.640, Z 61.200}
   LaserEnd_Ext()
   LIN {X 7.522, Y 15.640, Z 61.200}
   LaserStart_Ext()
   LIN {X -1.174, Y 15.640, Z 61.200}
   LaserEnd_Ext()
   LIN {X -1.250, Y 16.640, Z 61.200}
   LaserStart_Ext()
   LIN {X 7.332, Y 16.640, Z 61.200}
   LaserEnd_Ext()
   LIN {X 7.142, Y 17.640, Z 61.200}
   LaserStart_Ext()
   LIN {X -1.333, Y 17.640, Z 61.200}
   LaserEnd_Ext()
   LIN {X -1.415, Y 18.640, Z 61.200}
   LaserStart_Ext()
   LIN {X 6.952, Y 18.640, Z 61.200}
   LaserEnd_Ext()
   LIN {X 6.762, Y 19.640, Z 61.200}
   LaserStart_Ext()
   LIN {X -1.498, Y 19.640, Z 61.200}
   LaserEnd_Ext()
   LIN {X -1.580, Y 20.640, Z 61.200}
   LaserStart_Ext()
   LIN {X 6.572, Y 20.640, Z 61.200}
   LaserEnd_Ext()
   LIN {X 6.378, Y 21.640, Z 61.200}
   LaserStart_Ext()
   LIN {X -1.663, Y 21.640, Z 61.200}
   LaserEnd_Ext()
   LIN {X -1.746, Y 22.640, Z 61.200}
   LaserStart_Ext()
   LIN {X 6.122, Y 22.640, Z 61.200}
   LaserEnd_Ext()
   LIN {X 5.866, Y 23.640, Z 61.200}
   LaserStart_Ext()
   LIN {X -1.831, Y 23.640, Z 61.200}
   LaserEnd_Ext()
   LIN {X -2.012, Y 24.640, Z 61.200}
   LaserStart_Ext()
   LIN {X 5.609, Y 24.640, Z 61.200}
   LaserEnd_Ext()
   LIN {X 5.353, Y 25.640, Z 61.200}
   LaserStart_Ext()
   LIN {X -2.195, Y 25.640, Z 61.200}
   LaserEnd_Ext()
   LIN {X -2.378, Y 26.640, Z 61.200}
   LaserStart_Ext()
   LIN {X 5.076, Y 26.640, Z 61.200}
   LaserEnd_Ext()
   LIN {X 4.769, Y 27.640, Z 61.200}
   LaserStart_Ext()
   LIN {X -2.557, Y 27.640, Z 61.200}
   LaserEnd_Ext()
   LIN {X -2.736, Y 28.640, Z 61.200}
   LaserStart_Ext()
   LIN {X 4.462, Y 28.640, Z 61.200}
   LaserEnd_Ext()
   LIN {X 4.148, Y 29.640, Z 61.200}
   LaserStart_Ext()
   LIN {X -2.974, Y 29.640, Z 61.200}
   LaserEnd_Ext()
   LIN {X -3.214, Y 30.640, Z 61.200}
   LaserStart_Ext()
   LIN {X 3.832, Y 30.640, Z 61.200}
   LaserEnd_Ext()
   LIN {X 3.515, Y 31.640, Z 61.200}
   LaserStart_Ext()
   LIN {X -3.454, Y 31.640, Z 61.200}
   LaserEnd_Ext()
   LIN {X -3.738, Y 32.640, Z 61.200}
   LaserStart_Ext()
   LIN {X 3.199, Y 32.640, Z 61.200}
   LaserEnd_Ext()
   LIN {X 2.833, Y 33.640, Z 61.200}
   LaserStart_Ext()
   LIN {X -4.025, Y 33.640, Z 61.200}
   LaserEnd_Ext()
   LIN {X -4.310, Y 34.640, Z 61.200}
   LaserStart_Ext()
   LIN {X 2.465, Y 34.640, Z 61.200}
   LaserEnd_Ext()
   LIN {X 2.100, Y 35.640, Z 61.200}
   LaserStart_Ext()
   LIN {X -4.626, Y 35.640, Z 61.200}
   LaserEnd_Ext()
   LIN {X -4.955, Y 36.640, Z 61.200}
   LaserStart_Ext()
   LIN {X 1.718, Y 36.640, Z 61.200}
   LaserEnd_Ext()
   LIN {X 1.319, Y 37.640, Z 61.200}
   LaserStart_Ext()
   LIN {X -5.297, Y 37.640, Z 61.200}
   LaserEnd_Ext()
   LIN {X -5.656, Y 38.640, Z 61.200}
   LaserStart_Ext()
   LIN {X 0.917, Y 38.640, Z 61.200}
   LaserEnd_Ext()
   LIN {X 0.492, Y 39.640, Z 61.200}
   LaserStart_Ext()
   LIN {X -6.030, Y 39.640, Z 61.200}
   LaserEnd_Ext()
   LIN {X -6.278, Y 40.640, Z 61.200}
   LaserStart_Ext()
   LIN {X 0.066, Y 40.640, Z 61.200}
   LaserEnd_Ext()
   LIN {X -0.380, Y 41.640, Z 61.200}
   LaserStart_Ext()
   LIN {X -6.236, Y 41.640, Z 61.200}
   LaserEnd_Ext()
   LIN {X -5.779, Y 42.640, Z 61.200}
   LaserStart_Ext()
   LIN {X -0.950, Y 42.640, Z 61.200}
   LaserEnd_Ext()
   LIN {X -2.133, Y 43.640, Z 61.200}
   LaserStart_Ext()
   LIN {X -4.259, Y 43.640, Z 61.200}
   LaserEnd_Ext()
   LIN {X 1.109, Y -15.628, Z 62.050}
   LaserStart_Ext()
   LIN {X 1.478, Y -15.669, Z 62.050} C_DIS
   LIN {X 1.741, Y -15.827, Z 62.050} C_DIS
   LIN {X 3.304, Y -16.755, Z 62.050} C_DIS
   LIN {X 4.582, Y -18.781, Z 62.050} C_DIS
   LIN {X 4.660, Y -18.906, Z 62.050} C_DIS
   LIN {X 4.670, Y -19.042, Z 62.050} C_DIS
   LIN {X 4.834, Y -21.110, Z 62.050} C_DIS
   LIN {X 4.398, Y -22.170, Z 62.050} C_DIS
   LIN {X 3.889, Y -23.393, Z 62.050} C_DIS
   LIN {X 2.647, Y -24.512, Z 62.050} C_DIS
   LIN {X 2.386, Y -24.746, Z 62.050} C_DIS
   LIN {X 1.842, Y -24.918, Z 62.050} C_DIS
   LIN {X 0.305, Y -25.410, Z 62.050} C_DIS
   LIN {X -0.709, Y -25.299, Z 62.050} C_DIS
   LIN {X -1.729, Y -25.183, Z 62.050} C_DIS
   LIN {X -2.913, Y -24.484, Z 62.050} C_DIS
   LIN {X -3.509, Y -24.134, Z 62.050} C_DIS
   LIN {X -3.824, Y -23.698, Z 62.050} C_DIS
   LIN {X -4.722, Y -22.441, Z 62.050} C_DIS
   LIN {X -5.039, Y -20.825, Z 62.050} C_DIS
   LIN {X -5.126, Y -20.394, Z 62.050} C_DIS
   LIN {X -4.406, Y -18.132, Z 62.050} C_DIS
   LIN {X -4.236, Y -17.608, Z 62.050} C_DIS
   LIN {X -3.519, Y -16.939, Z 62.050} C_DIS
   LIN {X -2.664, Y -16.131, Z 62.050} C_DIS
   LIN {X -1.837, Y -15.861, Z 62.050} C_DIS
   LIN {X -0.552, Y -15.445, Z 62.050} C_DIS
   LIN {X 1.109, Y -15.628, Z 62.050}
   LaserEnd_Ext()
   LIN {X -6.094, Y -11.074, Z 62.050}
   LaserStart_Ext()
   LIN {X -7.200, Y -14.073, Z 62.050} C_DIS
   LIN {X -8.250, Y -16.566, Z 62.050} C_DIS
   LIN {X -8.352, Y -16.804, Z 62.050} C_DIS
   LIN {X -8.429, Y -17.110, Z 62.050} C_DIS
   LIN {X -9.116, Y -19.881, Z 62.050} C_DIS
   LIN {X -8.663, Y -23.093, Z 62.050} C_DIS
   LIN {X -8.599, Y -23.555, Z 62.050} C_DIS
   LIN {X -8.407, Y -23.867, Z 62.050} C_DIS
   LIN {X -6.610, Y -26.733, Z 62.050} C_DIS
   LIN {X -5.219, Y -27.766, Z 62.050} C_DIS
   LIN {X -4.271, Y -28.460, Z 62.050} C_DIS
   LIN {X -0.951, Y -29.239, Z 62.050} C_DIS
   LIN {X 0.146, Y -29.411, Z 62.050} C_DIS
   LIN {X 2.419, Y -29.050, Z 62.050} C_DIS
   LIN {X 4.723, Y -27.897, Z 62.050} C_DIS
   LIN {X 5.347, Y -27.558, Z 62.050} C_DIS
   LIN {X 6.200, Y -26.547, Z 62.050} C_DIS
   LIN {X 7.812, Y -24.656, Z 62.050} C_DIS
   LIN {X 8.271, Y -23.340, Z 62.050} C_DIS
   LIN {X 8.772, Y -21.872, Z 62.050} C_DIS
   LIN {X 9.151, Y -19.379, Z 62.050} C_DIS
   LIN {X 9.266, Y -18.646, Z 62.050} C_DIS
   LIN {X 9.330, Y -18.152, Z 62.050} C_DIS
   LIN {X 9.633, Y -15.708, Z 62.050} C_DIS
   LIN {X 9.879, Y -13.161, Z 62.050} C_DIS
   LIN {X 9.990, Y -11.919, Z 62.050} C_DIS
   LIN {X 10.202, Y -8.003, Z 62.050} C_DIS
   LIN {X 10.252, Y -7.138, Z 62.050} C_DIS
   LIN {X 10.257, Y -6.661, Z 62.050} C_DIS
   LIN {X 10.276, Y -0.624, Z 62.050} C_DIS
   LIN {X 10.251, Y 0.141, Z 62.050} C_DIS
   LIN {X 9.933, Y 5.595, Z 62.050} C_DIS
   LIN {X 9.727, Y 7.770, Z 62.050} C_DIS
   LIN {X 8.484, Y 16.039, Z 62.050} C_DIS
   LIN {X 7.491, Y 21.261, Z 62.050} C_DIS
   LIN {X 6.071, Y 26.800, Z 62.050} C_DIS
   LIN {X 4.137, Y 32.920, Z 62.050} C_DIS
   LIN {X 2.875, Y 36.350, Z 62.050} C_DIS
   LIN {X 1.783, Y 39.074, Z 62.050} C_DIS
   LIN {X 1.729, Y 39.199, Z 62.050} C_DIS
   LIN {X 0.850, Y 41.248, Z 62.050} C_DIS
   LIN {X 0.456, Y 42.127, Z 62.050} C_DIS
   LIN {X 0.198, Y 42.697, Z 62.050} C_DIS
   LIN {X -0.219, Y 43.287, Z 62.050} C_DIS
   LIN {X -0.649, Y 43.900, Z 62.050} C_DIS
   LIN {X -1.303, Y 44.307, Z 62.050} C_DIS
   LIN {X -2.128, Y 44.817, Z 62.050} C_DIS
   LIN {X -3.514, Y 44.980, Z 62.050} C_DIS
   LIN {X -3.861, Y 45.021, Z 62.050} C_DIS
   LIN {X -5.518, Y 44.223, Z 62.050} C_DIS
   LIN {X -6.273, Y 43.860, Z 62.050} C_DIS
   LIN {X -7.207, Y 42.339, Z 62.050} C_DIS
   LIN {X -7.320, Y 41.697, Z 62.050} C_DIS
   LIN {X -7.416, Y 40.955, Z 62.050} C_DIS
   LIN {X -7.251, Y 40.180, Z 62.050} C_DIS
   LIN {X -7.131, Y 39.599, Z 62.050} C_DIS
   LIN {X -6.970, Y 39.174, Z 62.050} C_DIS
   LIN {X -6.690, Y 38.428, Z 62.050} C_DIS
   LIN {X -6.208, Y 37.100, Z 62.050} C_DIS
   LIN {X -6.145, Y 36.924, Z 62.050} C_DIS
   LIN {X -6.011, Y 36.515, Z 62.050} C_DIS
   LIN {X -5.399, Y 34.673, Z 62.050} C_DIS
   LIN {X -4.823, Y 32.686, Z 62.050} C_DIS
   LIN {X -4.482, Y 31.497, Z 62.050} C_DIS
   LIN {X -4.053, Y 29.710, Z 62.050} C_DIS
   LIN {X -3.720, Y 28.335, Z 62.050} C_DIS
   LIN {X -3.466, Y 26.984, Z 62.050} C_DIS
   LIN {X -2.878, Y 23.767, Z 62.050} C_DIS
   LIN {X -2.402, Y 18.005, Z 62.050} C_DIS
   LIN {X -2.115, Y 14.632, Z 62.050} C_DIS
   LIN {X -2.062, Y 14.137, Z 62.050} C_DIS
   LIN {X -2.066, Y 13.625, Z 62.050} C_DIS
   LIN {X -2.108, Y 12.540, Z 62.050} C_DIS
   LIN {X -2.381, Y 5.832, Z 62.050} C_DIS
   LIN {X -3.067, Y 1.038, Z 62.050} C_DIS
   LIN {X -3.276, Y -0.498, Z 62.050} C_DIS
   LIN {X -3.709, Y -2.392, Z 62.050} C_DIS
   LIN {X -4.745, Y -6.809, Z 62.050} C_DIS
   LIN {X -5.682, Y -9.834, Z 62.050} C_DIS
   LIN {X -5.878, Y -10.478, Z 62.050} C_DIS
   LIN {X -6.094, Y -11.074, Z 62.050}
   LaserEnd_Ext()
   LIN {X 8.602, Y 8.528, Z 62.050}
   LaserStart_Ext()
   LIN {X 8.602, Y -15.898, Z 62.050}
   LaserEnd_Ext()
   LIN {X 7.602, Y -22.204, Z 62.050}
   LaserStart_Ext()
   LIN {X 7.602, Y 15.178, Z 62.050}
   LaserEnd_Ext()
   LIN {X 6.602, Y 20.583, Z 62.050}
   LaserStart_Ext()
   LIN {X 6.602, Y -24.534, Z 62.050}
   LaserEnd_Ext()
   LIN {X 5.602, Y -25.707, Z 62.050}
   LaserStart_Ext()
   LIN {X 5.602, Y -21.871, Z 62.050}
   LaserEnd_Ext()
   LIN {X 5.602, Y -18.573, Z 62.050}
   LaserStart_Ext()
   LIN {X 5.602, Y 24.604, Z 62.050}
   LaserEnd_Ext()
   LIN {X 4.602, Y 28.136, Z 62.050}
   LaserStart_Ext()
   LIN {X 4.602, Y -16.938, Z 62.050}
   LaserEnd_Ext()
   LIN {X 4.602, Y -24.093, Z 62.050}
   LaserStart_Ext()
   LIN {X 4.602, Y -26.825, Z 62.050}
   LaserEnd_Ext()
   LIN {X 3.602, Y -27.340, Z 62.050}
   LaserStart_Ext()
   LIN {X 3.602, Y -24.998, Z 62.050}
   LaserEnd_Ext()
   LIN {X 3.602, Y -15.769, Z 62.050}
   LaserStart_Ext()
   LIN {X 3.602, Y 31.297, Z 62.050}
   LaserEnd_Ext()
   LIN {X 2.602, Y 34.196, Z 62.050}
   LaserStart_Ext()
   LIN {X 2.602, Y -15.175, Z 62.050}
   LaserEnd_Ext()
   LIN {X 2.602, Y -25.726, Z 62.050}
   LaserStart_Ext()
   LIN {X 2.602, Y -27.840, Z 62.050}
   LaserEnd_Ext()
   LIN {X 1.602, Y -28.167, Z 62.050}
   LaserStart_Ext()
   LIN {X 1.602, Y -26.045, Z 62.050}
   LaserEnd_Ext()
   LIN {X 1.602, Y -14.678, Z 62.050}
   LaserStart_Ext()
   LIN {X 1.602, Y 36.838, Z 62.050}
   LaserEnd_Ext()
   LIN {X 0.602, Y 39.290, Z 62.050}
   LaserStart_Ext()
   LIN {X 0.602, Y -14.566, Z 62.050}
   LaserEnd_Ext()
   LIN {X 0.602, Y -26.365, Z 62.050}
   LaserStart_Ext()
   LIN {X 0.602, Y -28.326, Z 62.050}
   LaserEnd_Ext()
   LIN {X -0.398, Y -28.314, Z 62.050}
   LaserStart_Ext()
   LIN {X -0.398, Y -26.339, Z 62.050}
   LaserEnd_Ext()
   LIN {X -0.398, Y -14.456, Z 62.050}
   LaserStart_Ext()
   LIN {X -0.398, Y 41.587, Z 62.050}
   LaserEnd_Ext()
   LIN {X -1.398, Y 43.188, Z 62.050}
   LaserStart_Ext()
   LIN {X -1.398, Y 18.001, Z 62.050}
   LaserEnd_Ext()
   LIN {X -1.398, Y 5.641, Z 62.050}
   LaserStart_Ext()
   LIN {X -1.398, Y -14.668, Z 62.050}
   LaserEnd_Ext()
   LIN {X -1.398, Y -26.227, Z 62.050}
   LaserStart_Ext()
   LIN {X -1.398, Y -28.107, Z 62.050}
   LaserEnd_Ext()
   LIN {X -2.398, Y -27.872, Z 62.050}
   LaserStart_Ext()
   LIN {X -2.398, Y -25.949, Z 62.050}
   LaserEnd_Ext()
   LIN {X -2.398, Y -14.992, Z 62.050}
   LaserStart_Ext()
   LIN {X -2.398, Y -1.143, Z 62.050}
   LaserEnd_Ext()
   LIN {X -2.398, Y 26.703, Z 62.050}
   LaserStart_Ext()
   LIN {X -2.398, Y 43.809, Z 62.050}
   LaserEnd_Ext()
   LIN {X -3.398, Y 43.959, Z 62.050}
   LaserStart_Ext()
   LIN {X -3.398, Y 31.267, Z 62.050}
   LaserEnd_Ext()
   LIN {X -3.398, Y -5.444, Z 62.050}
   LaserStart_Ext()
   LIN {X -3.398, Y -15.448, Z 62.050}
   LaserEnd_Ext()
   LIN {X -3.398, Y -25.359, Z 62.050}
   LaserStart_Ext()
   LIN {X -3.398, Y -27.637, Z 62.050}
   LaserEnd_Ext()
   LIN {X -4.398, Y -27.127, Z 62.050}
   LaserStart_Ext()
   LIN {X -4.398, Y -24.611, Z 62.050}
   LaserEnd_Ext()
   LIN {X -4.398, Y -16.391, Z 62.050}
   LaserStart_Ext()
   LIN {X -4.398, Y -9.068, Z 62.050}
   LaserEnd_Ext()
   LIN {X -4.398, Y 34.811, Z 62.050}
   LaserStart_Ext()
   LIN {X -4.398, Y 43.652, Z 62.050}
   LaserEnd_Ext()
   LIN {X -5.398, Y 43.171, Z 62.050}
   LaserStart_Ext()
   LIN {X -5.398, Y 37.799, Z 62.050}
   LaserEnd_Ext()
   LIN {X -5.398, Y -12.077, Z 62.050}
   LaserStart_Ext()
   LIN {X -5.398, Y -17.951, Z 62.050}
   LaserEnd_Ext()
   LIN {X -5.398, Y -23.214, Z 62.050}
   LaserStart_Ext()
   LIN {X -5.398, Y -26.387, Z 62.050}
   LaserEnd_Ext()
   LIN {X -6.398, Y -25.188, Z 62.050}
   LaserStart_Ext()
   LIN {X -6.398, Y -14.746, Z 62.050}
   LaserEnd_Ext()
   LIN {X -6.398, Y 40.974, Z 62.050}
   LaserStart_Ext()
   LIN {X -6.398, Y 41.030, Z 62.050}
   LaserEnd_Ext()
   LIN {X -7.398, Y -17.117, Z 62.050}
   LaserStart_Ext()
   LIN {X -7.398, Y -23.593, Z 62.050}
   LaserEnd_Ext()
   LIN {X 4.132, Y -22.946, Z 62.900}
   LaserStart_Ext()
   LIN {X 3.968, Y -23.340, Z 62.900} C_DIS
   LIN {X 3.373, Y -23.876, Z 62.900} C_DIS
   LIN {X 2.449, Y -24.702, Z 62.900} C_DIS
   LIN {X 1.595, Y -24.973, Z 62.900} C_DIS
   LIN {X 0.395, Y -25.357, Z 62.900} C_DIS
   LIN {X -1.288, Y -25.172, Z 62.900} C_DIS
   LIN {X -1.639, Y -25.134, Z 62.900} C_DIS
   LIN {X -1.862, Y -25.005, Z 62.900} C_DIS
   LIN {X -3.422, Y -24.090, Z 62.900} C_DIS
   LIN {X -4.522, Y -22.563, Z 62.900} C_DIS
   LIN {X -4.639, Y -22.399, Z 62.900} C_DIS
   LIN {X -4.680, Y -22.189, Z 62.900} C_DIS
   LIN {X -5.047, Y -20.353, Z 62.900} C_DIS
   LIN {X -4.627, Y -19.032, Z 62.900} C_DIS
   LIN {X -4.141, Y -17.531, Z 62.900} C_DIS
   LIN {X -2.907, Y -16.380, Z 62.900} C_DIS
   LIN {X -2.573, Y -16.071, Z 62.900} C_DIS
   LIN {X -1.935, Y -15.863, Z 62.900} C_DIS
   LIN {X -0.486, Y -15.394, Z 62.900} C_DIS
   LIN {X 0.555, Y -15.508, Z 62.900} C_DIS
   LIN {X 1.545, Y -15.613, Z 62.900} C_DIS
   LIN {X 2.668, Y -16.275, Z 62.900} C_DIS
   LIN {X 3.374, Y -16.695, Z 62.900} C_DIS
   LIN {X 3.844, Y -17.440, Z 62.900} C_DIS
   LIN {X 4.735, Y -18.842, Z 62.900} C_DIS
   LIN {X 4.857, Y -20.328, Z 62.900} C_DIS
   LIN {X 4.914, Y -21.046, Z 62.900} C_DIS
   LIN {X 4.132, Y -22.946, Z 62.900}
   LaserEnd_Ext()
   LIN {X -7.199, Y 42.582, Z 62.900}
   LaserStart_Ext()
   LIN {X -6.907, Y 43.061, Z 62.900} C_DIS
   LIN {X -6.310, Y 43.933, Z 62.900} C_DIS
   LIN {X -5.164, Y 44.484, Z 62.900} C_DIS
   LIN {X -3.936, Y 45.064, Z 62.900} C_DIS
   LIN {X -2.804, Y 44.935, Z 62.900} C_DIS
   LIN {X -2.202, Y 44.865, Z 62.900} C_DIS
   LIN {X -1.483, Y 44.419, Z 62.900} C_DIS
   LIN {X -0.722, Y 43.950, Z 62.900} C_DIS
   LIN {X -0.359, Y 43.440, Z 62.900} C_DIS
   LIN {X 0.128, Y 42.749, Z 62.900} C_DIS
   LIN {X 0.599, Y 41.710, Z 62.900} C_DIS
   LIN {X 0.769, Y 41.336, Z 62.900} C_DIS
   LIN {X 0.926, Y 40.976, Z 62.900} C_DIS
   LIN {X 1.670, Y 39.252, Z 62.900} C_DIS
   LIN {X 2.227, Y 37.863, Z 62.900} C_DIS
   LIN {X 2.487, Y 37.212, Z 62.900} C_DIS
   LIN {X 2.770, Y 36.532, Z 62.900} C_DIS
   LIN {X 3.199, Y 35.398, Z 62.900} C_DIS
   LIN {X 4.141, Y 32.837, Z 62.900} C_DIS
   LIN {X 5.572, Y 28.316, Z 62.900} C_DIS
   LIN {X 6.053, Y 26.827, Z 62.900} C_DIS
   LIN {X 6.534, Y 24.930, Z 62.900} C_DIS
   LIN {X 7.615, Y 20.713, Z 62.900} C_DIS
   LIN {X 8.370, Y 16.739, Z 62.900} C_DIS
   LIN {X 9.815, Y 7.127, Z 62.900} C_DIS
   LIN {X 9.943, Y 5.780, Z 62.900} C_DIS
   LIN {X 10.303, Y -0.393, Z 62.900} C_DIS
   LIN {X 10.308, Y -0.547, Z 62.900} C_DIS
   LIN {X 10.303, Y -2.122, Z 62.900} C_DIS
   LIN {X 10.299, Y -7.061, Z 62.900} C_DIS
   LIN {X 10.238, Y -8.350, Z 62.900} C_DIS
   LIN {X 10.048, Y -11.842, Z 62.900} C_DIS
   LIN {X 9.823, Y -14.365, Z 62.900} C_DIS
   LIN {X 9.701, Y -15.632, Z 62.900} C_DIS
   LIN {X 9.474, Y -17.461, Z 62.900} C_DIS
   LIN {X 9.340, Y -18.572, Z 62.900} C_DIS
   LIN {X 9.235, Y -19.293, Z 62.900} C_DIS
   LIN {X 8.854, Y -21.799, Z 62.900} C_DIS
   LIN {X 7.983, Y -24.348, Z 62.900} C_DIS
   LIN {X 7.902, Y -24.583, Z 62.900} C_DIS
   LIN {X 7.614, Y -24.920, Z 62.900} C_DIS
   LIN {X 5.444, Y -27.490, Z 62.900} C_DIS
   LIN {X 3.858, Y -28.355, Z 62.900} C_DIS
   LIN {X 2.686, Y -28.941, Z 62.900} C_DIS
   LIN {X 1.167, Y -29.183, Z 62.900} C_DIS
   LIN {X -0.034, Y -29.389, Z 62.900} C_DIS
   LIN {X -4.173, Y -28.417, Z 62.900} C_DIS
   LIN {X -5.971, Y -27.101, Z 62.900} C_DIS
   LIN {X -6.517, Y -26.696, Z 62.900} C_DIS
   LIN {X -7.442, Y -25.221, Z 62.900} C_DIS
   LIN {X -8.514, Y -23.523, Z 62.900} C_DIS
   LIN {X -8.730, Y -22.036, Z 62.900} C_DIS
   LIN {X -9.039, Y -19.850, Z 62.900} C_DIS
   LIN {X -8.599, Y -18.076, Z 62.900} C_DIS
   LIN {X -8.282, Y -16.771, Z 62.900} C_DIS
   LIN {X -7.741, Y -15.473, Z 62.900} C_DIS
   LIN {X -7.136, Y -14.038, Z 62.900} C_DIS
   LIN {X -6.615, Y -12.625, Z 62.900} C_DIS
   LIN {X -5.822, Y -10.436, Z 62.900} C_DIS
   LIN {X -5.102, Y -8.068, Z 62.900} C_DIS
   LIN {X -4.697, Y -6.762, Z 62.900} C_DIS
   LIN {X -4.250, Y -4.855, Z 62.900} C_DIS
   LIN {X -3.249, Y -0.479, Z 62.900} C_DIS
   LIN {X -2.764, Y 3.073, Z 62.900} C_DIS
   LIN {X -2.368, Y 5.841, Z 62.900} C_DIS
   LIN {X -2.210, Y 9.715, Z 62.900} C_DIS
   LIN {X -2.089, Y 12.866, Z 62.900} C_DIS
   LIN {X -2.077, Y 14.353, Z 62.900} C_DIS
   LIN {X -2.230, Y 15.793, Z 62.900} C_DIS
   LIN {X -2.927, Y 23.978, Z 62.900} C_DIS
   LIN {X -2.970, Y 24.195, Z 62.900} C_DIS
   LIN {X -3.034, Y 24.534, Z 62.900} C_DIS
   LIN {X -3.757, Y 28.383, Z 62.900} C_DIS
   LIN {X -4.318, Y 30.701, Z 62.900} C_DIS
   LIN {X -4.564, Y 31.678, Z 62.900} C_DIS
   LIN {X -5.109, Y 33.539, Z 62.900} C_DIS
   LIN {X -5.450, Y 34.713, Z 62.900} C_DIS
   LIN {X -5.658, Y 35.338, Z 62.900} C_DIS
   LIN {X -6.201, Y 36.962, Z 62.900} C_DIS
   LIN {X -6.727, Y 38.404, Z 62.900} C_DIS
   LIN {X -6.781, Y 38.550, Z 62.900} C_DIS
   LIN {X -7.193, Y 39.634, Z 62.900} C_DIS
   LIN {X -7.405, Y 40.657, Z 62.900} C_DIS
   LIN {X -7.483, Y 41.038, Z 62.900} C_DIS
   LIN {X -7.376, Y 41.580, Z 62.900} C_DIS
   LIN {X -7.199, Y 42.582, Z 62.900}
   LaserEnd_Ext()
   LIN {X -4.857, Y 43.522, Z 62.900}
   LaserStart_Ext()
   LIN {X -1.932, Y 43.522, Z 62.900}
   LaserEnd_Ext()
   LIN {X -0.935, Y 42.522, Z 62.900}
   LaserStart_Ext()
   LIN {X -6.064, Y 42.522, Z 62.900}
   LaserEnd_Ext()
   LIN {X -6.371, Y 41.522, Z 62.900}
   LaserStart_Ext()
   LIN {X -0.414, Y 41.522, Z 62.900}
   LaserEnd_Ext()
   LIN {X 0.033, Y 40.522, Z 62.900}
   LaserStart_Ext()
   LIN {X -6.356, Y 40.522, Z 62.900}
   LaserEnd_Ext()
   LIN {X -6.081, Y 39.522, Z 62.900}
   LaserStart_Ext()
   LIN {X 0.464, Y 39.522, Z 62.900}
   LaserEnd_Ext()
   LIN {X 0.885, Y 38.522, Z 62.900}
   LaserStart_Ext()
   LIN {X -5.705, Y 38.522, Z 62.900}
   LaserEnd_Ext()
   LIN {X -5.341, Y 37.522, Z 62.900}
   LaserStart_Ext()
   LIN {X 1.286, Y 37.522, Z 62.900}
   LaserEnd_Ext()
   LIN {X 1.691, Y 36.522, Z 62.900}
   LaserStart_Ext()
   LIN {X -4.999, Y 36.522, Z 62.900}
   LaserEnd_Ext()
   LIN {X -4.665, Y 35.522, Z 62.900}
   LaserStart_Ext()
   LIN {X 2.083, Y 35.522, Z 62.900}
   LaserEnd_Ext()
   LIN {X 2.456, Y 34.522, Z 62.900}
   LaserStart_Ext()
   LIN {X -4.353, Y 34.522, Z 62.900}
   LaserEnd_Ext()
   LIN {X -4.062, Y 33.522, Z 62.900}
   LaserStart_Ext()
   LIN {X 2.824, Y 33.522, Z 62.900}
   LaserEnd_Ext()
   LIN {X 3.192, Y 32.522, Z 62.900}
   LaserStart_Ext()
   LIN {X -3.769, Y 32.522, Z 62.900}
   LaserEnd_Ext()
   LIN {X -3.493, Y 31.522, Z 62.900}
   LaserStart_Ext()
   LIN {X 3.509, Y 31.522, Z 62.900}
   LaserEnd_Ext()
   LIN {X 3.825, Y 30.522, Z 62.900}
   LaserStart_Ext()
   LIN {X -3.246, Y 30.522, Z 62.900}
   LaserEnd_Ext()
   LIN {X -3.004, Y 29.522, Z 62.900}
   LaserStart_Ext()
   LIN {X 4.141, Y 29.522, Z 62.900}
   LaserEnd_Ext()
   LIN {X 4.458, Y 28.522, Z 62.900}
   LaserStart_Ext()
   LIN {X -2.765, Y 28.522, Z 62.900}
   LaserEnd_Ext()
   LIN {X -2.577, Y 27.522, Z 62.900}
   LaserStart_Ext()
   LIN {X 4.777, Y 27.522, Z 62.900}
   LaserEnd_Ext()
   LIN {X 5.098, Y 26.522, Z 62.900}
   LaserStart_Ext()
   LIN {X -2.390, Y 26.522, Z 62.900}
   LaserEnd_Ext()
   LIN {X -2.202, Y 25.522, Z 62.900}
   LaserStart_Ext()
   LIN {X 5.352, Y 25.522, Z 62.900}
   LaserEnd_Ext()
   LIN {X 5.606, Y 24.522, Z 62.900}
   LaserStart_Ext()
   LIN {X -2.014, Y 24.522, Z 62.900}
   LaserEnd_Ext()
   LIN {X -1.885, Y 23.522, Z 62.900}
   LaserStart_Ext()
   LIN {X 5.862, Y 23.522, Z 62.900}
   LaserEnd_Ext()
   LIN {X 6.119, Y 22.522, Z 62.900}
   LaserStart_Ext()
   LIN {X -1.799, Y 22.522, Z 62.900}
   LaserEnd_Ext()
   LIN {X -1.714, Y 21.522, Z 62.900}
   LaserStart_Ext()
   LIN {X 6.375, Y 21.522, Z 62.900}
   LaserEnd_Ext()
   LIN {X 6.631, Y 20.522, Z 62.900}
   LaserStart_Ext()
   LIN {X -1.629, Y 20.522, Z 62.900}
   LaserEnd_Ext()
   LIN {X -1.544, Y 19.522, Z 62.900}
   LaserStart_Ext()
   LIN {X 6.823, Y 19.522, Z 62.900}
   LaserEnd_Ext()
   LIN {X 7.013, Y 18.522, Z 62.900}
   LaserStart_Ext()
   LIN {X -1.459, Y 18.522, Z 62.900}
   LaserEnd_Ext()
   LIN {X -1.373, Y 17.522, Z 62.900}
   LaserStart_Ext()
   LIN {X 7.203, Y 17.522, Z 62.900}
   LaserEnd_Ext()
   LIN {X 7.392, Y 16.522, Z 62.900}
   LaserStart_Ext()
   LIN {X -1.288, Y 16.522, Z 62.900}
   LaserEnd_Ext()
   LIN {X -1.195, Y 15.522, Z 62.900}
   LaserStart_Ext()
   LIN {X 7.542, Y 15.522, Z 62.900}
   LaserEnd_Ext()
   LIN {X 7.692, Y 14.522, Z 62.900}
   LaserStart_Ext()
   LIN {X -1.089, Y 14.522, Z 62.900}
   LaserEnd_Ext()
   LIN {X -1.084, Y 13.522, Z 62.900}
   LaserStart_Ext()
   LIN {X 7.843, Y 13.522, Z 62.900}
   LaserEnd_Ext()
   LIN {X 7.993, Y 12.522, Z 62.900}
   LaserStart_Ext()
   LIN {X -1.102, Y 12.522, Z 62.900}
   LaserEnd_Ext()
   LIN {X -1.140, Y 11.522, Z 62.900}
   LaserStart_Ext()
   LIN {X 8.143, Y 11.522, Z 62.900}
   LaserEnd_Ext()
   LIN {X 8.294, Y 10.522, Z 62.900}
   LaserStart_Ext()
   LIN {X -1.179, Y 10.522, Z 62.900}
   LaserEnd_Ext()
   LIN {X -1.217, Y 9.522, Z 62.900}
   LaserStart_Ext()
   LIN {X 8.444, Y 9.522, Z 62.900}
   LaserEnd_Ext()
   LIN {X 8.594, Y 8.522, Z 62.900}
   LaserStart_Ext()
   LIN {X -1.258, Y 8.522, Z 62.900}
   LaserEnd_Ext()
   LIN {X -1.299, Y 7.522, Z 62.900}
   LaserStart_Ext()
   LIN {X 8.745, Y 7.522, Z 62.900}
   LaserEnd_Ext()
   LIN {X 8.868, Y 6.522, Z 62.900}
   LaserStart_Ext()
   LIN {X -1.339, Y 6.522, Z 62.900}
   LaserEnd_Ext()
   LIN {X -1.403, Y 5.522, Z 62.900}
   LaserStart_Ext()
   LIN {X 8.956, Y 5.522, Z 62.900}
   LaserEnd_Ext()
   LIN {X 9.015, Y 4.522, Z 62.900}
   LaserStart_Ext()
   LIN {X -1.546, Y 4.522, Z 62.900}
   LaserEnd_Ext()
   LIN {X -1.690, Y 3.522, Z 62.900}
   LaserStart_Ext()
   LIN {X 9.073, Y 3.522, Z 62.900}
   LaserEnd_Ext()
   LIN {X 9.131, Y 2.522, Z 62.900}
   LaserStart_Ext()
   LIN {X -1.830, Y 2.522, Z 62.900}
   LaserEnd_Ext()
   LIN {X -1.966, Y 1.522, Z 62.900}
   LaserStart_Ext()
   LIN {X 9.189, Y 1.522, Z 62.900}
   LaserEnd_Ext()
   LIN {X 9.248, Y 0.522, Z 62.900}
   LaserStart_Ext()
   LIN {X -2.103, Y 0.522, Z 62.900}
   LaserEnd_Ext()
   LIN {X -2.240, Y -0.478, Z 62.900}
   LaserStart_Ext()
   LIN {X 9.305, Y -0.478, Z 62.900}
   LaserEnd_Ext()
   LIN {X 9.305, Y -1.478, Z 62.900}
   LaserStart_Ext()
   LIN {X -2.452, Y -1.478, Z 62.900}
   LaserEnd_Ext()
   LIN {X -2.681, Y -2.478, Z 62.900}
   LaserStart_Ext()
   LIN {X 9.302, Y -2.478, Z 62.900}
   LaserEnd_Ext()
   LIN {X 9.302, Y -3.478, Z 62.900}
   LaserStart_Ext()
   LIN {X -2.909, Y -3.478, Z 62.900}
   LaserEnd_Ext()
   LIN {X -3.138, Y -4.478, Z 62.900}
   LaserStart_Ext()
   LIN {X 9.301, Y -4.478, Z 62.900}
   LaserEnd_Ext()
   LIN {X 9.300, Y -5.478, Z 62.900}
   LaserStart_Ext()
   LIN {X -3.369, Y -5.478, Z 62.900}
   LaserEnd_Ext()
   LIN {X -3.604, Y -6.478, Z 62.900}
   LaserStart_Ext()
   LIN {X 9.300, Y -6.478, Z 62.900}
   LaserEnd_Ext()
   LIN {X 9.278, Y -7.478, Z 62.900}
   LaserStart_Ext()
   LIN {X -3.872, Y -7.478, Z 62.900}
   LaserEnd_Ext()
   LIN {X -4.181, Y -8.478, Z 62.900}
   LaserStart_Ext()
   LIN {X 9.230, Y -8.478, Z 62.900}
   LaserEnd_Ext()
   LIN {X 9.175, Y -9.478, Z 62.900}
   LaserStart_Ext()
   LIN {X -4.486, Y -9.478, Z 62.900}
   LaserEnd_Ext()
   LIN {X -4.790, Y -10.478, Z 62.900}
   LaserStart_Ext()
   LIN {X 9.121, Y -10.478, Z 62.900}
   LaserEnd_Ext()
   LIN {X 9.066, Y -11.478, Z 62.900}
   LaserStart_Ext()
   LIN {X -5.136, Y -11.478, Z 62.900}
   LaserEnd_Ext()
   LIN {X -5.499, Y -12.478, Z 62.900}
   LaserStart_Ext()
   LIN {X 8.987, Y -12.478, Z 62.900}
   LaserEnd_Ext()
   LIN {X 8.898, Y -13.478, Z 62.900}
   LaserStart_Ext()
   LIN {X -5.864, Y -13.478, Z 62.900}
   LaserEnd_Ext()
   LIN {X -6.237, Y -14.478, Z 62.900}
   LaserStart_Ext()
   LIN {X -0.904, Y -14.478, Z 62.900}
   LaserEnd_Ext()
   LIN {X 0.338, Y -14.478, Z 62.900}
   LaserStart_Ext()
   LIN {X 8.807, Y -14.478, Z 62.900}
   LaserEnd_Ext()
   LIN {X 8.711, Y -15.478, Z 62.900}
   LaserStart_Ext()
   LIN {X 3.284, Y -15.478, Z 62.900}
   LaserEnd_Ext()
   LIN {X -3.405, Y -15.478, Z 62.900}
   LaserStart_Ext()
   LIN {X -6.658, Y -15.478, Z 62.900}
   LaserEnd_Ext()
   LIN {X -7.077, Y -16.478, Z 62.900}
   LaserStart_Ext()
   LIN {X -4.478, Y -16.478, Z 62.900}
   LaserEnd_Ext()
   LIN {X 4.420, Y -16.478, Z 62.900}
   LaserStart_Ext()
   LIN {X 8.588, Y -16.478, Z 62.900}
   LaserEnd_Ext()
   LIN {X 8.464, Y -17.478, Z 62.900}
   LaserStart_Ext()
   LIN {X 5.053, Y -17.478, Z 62.900}
   LaserEnd_Ext()
   LIN {X -5.175, Y -17.478, Z 62.900}
   LaserStart_Ext()
   LIN {X -7.425, Y -17.478, Z 62.900}
   LaserEnd_Ext()
   LIN {X -7.669, Y -18.478, Z 62.900}
   LaserStart_Ext()
   LIN {X -5.499, Y -18.478, Z 62.900}
   LaserEnd_Ext()
   LIN {X 5.667, Y -18.478, Z 62.900}
   LaserStart_Ext()
   LIN {X 8.343, Y -18.478, Z 62.900}
   LaserEnd_Ext()
   LIN {X 8.195, Y -19.478, Z 62.900}
   LaserStart_Ext()
   LIN {X 5.791, Y -19.478, Z 62.900}
   LaserEnd_Ext()
   LIN {X -5.818, Y -19.478, Z 62.900}
   LaserStart_Ext()
   LIN {X -7.917, Y -19.478, Z 62.900}
   LaserEnd_Ext()
   LIN {X -7.941, Y -20.478, Z 62.900}
   LaserStart_Ext()
   LIN {X -6.038, Y -20.478, Z 62.900}
   LaserEnd_Ext()
   LIN {X 5.872, Y -20.478, Z 62.900}
   LaserStart_Ext()
   LIN {X 8.043, Y -20.478, Z 62.900}
   LaserEnd_Ext()
   LIN {X 7.891, Y -21.478, Z 62.900}
   LaserStart_Ext()
   LIN {X 5.817, Y -21.478, Z 62.900}
   LaserEnd_Ext()
   LIN {X -5.842, Y -21.478, Z 62.900}
   LaserStart_Ext()
   LIN {X -7.799, Y -21.478, Z 62.900}
   LaserEnd_Ext()
   LIN {X -7.655, Y -22.478, Z 62.900}
   LaserStart_Ext()
   LIN {X -5.642, Y -22.478, Z 62.900}
   LaserEnd_Ext()
   LIN {X 5.406, Y -22.478, Z 62.900}
   LaserStart_Ext()
   LIN {X 7.565, Y -22.478, Z 62.900}
   LaserEnd_Ext()
   LIN {X 7.224, Y -23.478, Z 62.900}
   LaserStart_Ext()
   LIN {X 4.994, Y -23.478, Z 62.900}
   LaserEnd_Ext()
   LIN {X -5.095, Y -23.478, Z 62.900}
   LaserStart_Ext()
   LIN {X -7.359, Y -23.478, Z 62.900}
   LaserEnd_Ext()
   LIN {X -6.728, Y -24.478, Z 62.900}
   LaserStart_Ext()
   LIN {X -4.374, Y -24.478, Z 62.900}
   LaserEnd_Ext()
   LIN {X 4.198, Y -24.478, Z 62.900}
   LaserStart_Ext()
   LIN {X 6.678, Y -24.478, Z 62.900}
   LaserEnd_Ext()
   LIN {X 5.834, Y -25.478, Z 62.900}
   LaserStart_Ext()
   LIN {X 3.077, Y -25.478, Z 62.900}
   LaserEnd_Ext()
   LIN {X -3.031, Y -25.478, Z 62.900}
   LaserStart_Ext()
   LIN {X -6.100, Y -25.478, Z 62.900}
   LaserEnd_Ext()
   LIN {X -5.129, Y -26.478, Z 62.900}
   LaserStart_Ext()
   LIN {X 4.990, Y -26.478, Z 62.900}
   LaserEnd_Ext()
   LIN {X 3.375, Y -27.478, Z 62.900}
   LaserStart_Ext()
   LIN {X -3.762, Y -27.478, Z 62.900}
   LaserEnd_Ext()
   LIN {X -4.555, Y -22.357, Z 63.750}
   LaserStart_Ext()
   LIN {X -4.837, Y -20.970, Z 63.750} C_DIS
   LIN {X -4.969, Y -20.312, Z 63.750} C_DIS
   LIN {X -4.848, Y -19.933, Z 63.750} C_DIS
   LIN {X -4.045, Y -17.454, Z 63.750} C_DIS
   LIN {X -3.770, Y -17.197, Z 63.750} C_DIS
   LIN {X -2.505, Y -16.024, Z 63.750} C_DIS
   LIN {X -0.663, Y -15.423, Z 63.750} C_DIS
   LIN {X -0.419, Y -15.342, Z 63.750} C_DIS
   LIN {X -0.113, Y -15.374, Z 63.750} C_DIS
   LIN {X 1.612, Y -15.557, Z 63.750} C_DIS
   LIN {X 2.847, Y -16.285, Z 63.750} C_DIS
   LIN {X 3.444, Y -16.634, Z 63.750} C_DIS
   LIN {X 3.984, Y -17.479, Z 63.750} C_DIS
   LIN {X 4.810, Y -18.779, Z 63.750} C_DIS
   LIN {X 4.916, Y -20.069, Z 63.750} C_DIS
   LIN {X 4.994, Y -20.981, Z 63.750} C_DIS
   LIN {X 4.820, Y -21.428, Z 63.750} C_DIS
   LIN {X 4.065, Y -23.262, Z 63.750} C_DIS
   LIN {X 3.527, Y -23.747, Z 63.750} C_DIS
   LIN {X 2.500, Y -24.665, Z 63.750} C_DIS
   LIN {X 0.518, Y -25.293, Z 63.750} C_DIS
   LIN {X -1.550, Y -25.085, Z 63.750} C_DIS
   LIN {X -2.860, Y -24.324, Z 63.750} C_DIS
   LIN {X -3.335, Y -24.045, Z 63.750} C_DIS
   LIN {X -3.749, Y -23.471, Z 63.750} C_DIS
   LIN {X -4.555, Y -22.357, Z 63.750}
   LaserEnd_Ext()
   LIN {X -2.355, Y 5.851, Z 63.750}
   LaserStart_Ext()
   LIN {X -2.313, Y 6.891, Z 63.750} C_DIS
   LIN {X -2.112, Y 12.107, Z 63.750} C_DIS
   LIN {X -2.092, Y 14.569, Z 63.750} C_DIS
   LIN {X -2.345, Y 16.953, Z 63.750} C_DIS
   LIN {X -2.942, Y 23.962, Z 63.750} C_DIS
   LIN {X -3.187, Y 25.204, Z 63.750} C_DIS
   LIN {X -3.552, Y 27.144, Z 63.750} C_DIS
   LIN {X -3.793, Y 28.430, Z 63.750} C_DIS
   LIN {X -3.981, Y 29.204, Z 63.750} C_DIS
   LIN {X -4.677, Y 31.975, Z 63.750} C_DIS
   LIN {X -5.192, Y 33.729, Z 63.750} C_DIS
   LIN {X -5.501, Y 34.753, Z 63.750} C_DIS
   LIN {X -6.054, Y 36.394, Z 63.750} C_DIS
   LIN {X -6.257, Y 36.999, Z 63.750} C_DIS
   LIN {X -6.362, Y 37.288, Z 63.750} C_DIS
   LIN {X -6.809, Y 38.501, Z 63.750} C_DIS
   LIN {X -7.149, Y 39.394, Z 63.750} C_DIS
   LIN {X -7.255, Y 39.670, Z 63.750} C_DIS
   LIN {X -7.359, Y 40.192, Z 63.750} C_DIS
   LIN {X -7.549, Y 41.123, Z 63.750} C_DIS
   LIN {X -7.378, Y 41.990, Z 63.750} C_DIS
   LIN {X -7.220, Y 42.742, Z 63.750} C_DIS
   LIN {X -6.485, Y 43.811, Z 63.750} C_DIS
   LIN {X -6.324, Y 44.026, Z 63.750} C_DIS
   LIN {X -5.193, Y 44.549, Z 63.750} C_DIS
   LIN {X -4.011, Y 45.107, Z 63.750} C_DIS
   LIN {X -3.478, Y 45.046, Z 63.750} C_DIS
   LIN {X -2.277, Y 44.912, Z 63.750} C_DIS
   LIN {X -1.588, Y 44.490, Z 63.750} C_DIS
   LIN {X -0.794, Y 44.001, Z 63.750} C_DIS
   LIN {X -0.252, Y 43.238, Z 63.750} C_DIS
   LIN {X 0.059, Y 42.802, Z 63.750} C_DIS
   LIN {X 0.247, Y 42.392, Z 63.750} C_DIS
   LIN {X 0.687, Y 41.423, Z 63.750} C_DIS
   LIN {X 1.522, Y 39.512, Z 63.750} C_DIS
   LIN {X 1.579, Y 39.377, Z 63.750} C_DIS
   LIN {X 2.099, Y 38.074, Z 63.750} C_DIS
   LIN {X 2.666, Y 36.715, Z 63.750} C_DIS
   LIN {X 3.523, Y 34.446, Z 63.750} C_DIS
   LIN {X 4.145, Y 32.754, Z 63.750} C_DIS
   LIN {X 5.090, Y 29.769, Z 63.750} C_DIS
   LIN {X 6.043, Y 26.818, Z 63.750} C_DIS
   LIN {X 6.996, Y 23.059, Z 63.750} C_DIS
   LIN {X 7.738, Y 20.166, Z 63.750} C_DIS
   LIN {X 8.256, Y 17.439, Z 63.750} C_DIS
   LIN {X 9.904, Y 6.484, Z 63.750} C_DIS
   LIN {X 9.953, Y 5.965, Z 63.750} C_DIS
   LIN {X 10.122, Y 3.070, Z 63.750} C_DIS
   LIN {X 10.340, Y -0.470, Z 63.750} C_DIS
   LIN {X 10.350, Y -2.140, Z 63.750} C_DIS
   LIN {X 10.347, Y -6.984, Z 63.750} C_DIS
   LIN {X 10.207, Y -9.914, Z 63.750} C_DIS
   LIN {X 10.107, Y -11.766, Z 63.750} C_DIS
   LIN {X 9.771, Y -15.526, Z 63.750} C_DIS
   LIN {X 9.415, Y -18.496, Z 63.750} C_DIS
   LIN {X 9.135, Y -20.417, Z 63.750} C_DIS
   LIN {X 8.936, Y -21.725, Z 63.750} C_DIS
   LIN {X 8.382, Y -23.347, Z 63.750} C_DIS
   LIN {X 7.989, Y -24.514, Z 63.750} C_DIS
   LIN {X 7.259, Y -25.389, Z 63.750} C_DIS
   LIN {X 5.541, Y -27.423, Z 63.750} C_DIS
   LIN {X 2.993, Y -28.812, Z 63.750} C_DIS
   LIN {X 0.018, Y -29.337, Z 63.750} C_DIS
   LIN {X -4.076, Y -28.374, Z 63.750} C_DIS
   LIN {X -5.753, Y -27.147, Z 63.750} C_DIS
   LIN {X -6.423, Y -26.659, Z 63.750} C_DIS
   LIN {X -6.697, Y -26.232, Z 63.750} C_DIS
   LIN {X -8.428, Y -23.490, Z 63.750} C_DIS
   LIN {X -8.936, Y -20.006, Z 63.750} C_DIS
   LIN {X -8.962, Y -19.819, Z 63.750} C_DIS
   LIN {X -8.924, Y -19.666, Z 63.750} C_DIS
   LIN {X -8.212, Y -16.738, Z 63.750} C_DIS
   LIN {X -7.129, Y -14.140, Z 63.750} C_DIS
   LIN {X -7.073, Y -14.002, Z 63.750} C_DIS
   LIN {X -6.989, Y -13.766, Z 63.750} C_DIS
   LIN {X -5.765, Y -10.393, Z 63.750} C_DIS
   LIN {X -4.796, Y -7.206, Z 63.750} C_DIS
   LIN {X -4.649, Y -6.715, Z 63.750} C_DIS
   LIN {X -4.571, Y -6.359, Z 63.750} C_DIS
   LIN {X -3.222, Y -0.459, Z 63.750} C_DIS
   LIN {X -2.461, Y 5.108, Z 63.750} C_DIS
   LIN {X -2.355, Y 5.851, Z 63.750}
   LaserEnd_Ext()
   LIN {X -7.280, Y -23.435, Z 63.750}
   LaserStart_Ext()
   LIN {X -7.280, Y -17.138, Z 63.750}
   LaserEnd_Ext()
   LIN {X -6.280, Y 42.345, Z 63.750}
   LaserStart_Ext()
   LIN {X -6.280, Y 39.920, Z 63.750}
   LaserEnd_Ext()
   LIN {X -6.280, Y -14.701, Z 63.750}
   LaserStart_Ext()
   LIN {X -6.280, Y -25.019, Z 63.750}
   LaserEnd_Ext()
   LIN {X -5.280, Y -26.254, Z 63.750}
   LaserStart_Ext()
   LIN {X -5.280, Y -23.062, Z 63.750}
   LaserEnd_Ext()
   LIN {X -5.280, Y -18.021, Z 63.750}
   LaserStart_Ext()
   LIN {X -5.280, Y -11.988, Z 63.750}
   LaserEnd_Ext()
   LIN {X -5.280, Y 37.230, Z 63.750}
   LaserStart_Ext()
   LIN {X -5.280, Y 43.407, Z 63.750}
   LaserEnd_Ext()
   LIN {X -4.280, Y 43.874, Z 63.750}
   LaserStart_Ext()
   LIN {X -4.280, Y 34.168, Z 63.750}
   LaserEnd_Ext()
   LIN {X -4.280, Y -8.945, Z 63.750}
   LaserStart_Ext()
   LIN {X -4.280, Y -16.307, Z 63.750}
   LaserEnd_Ext()
   LIN {X -4.280, Y -24.444, Z 63.750}
   LaserStart_Ext()
   LIN {X -4.280, Y -26.986, Z 63.750}
   LaserEnd_Ext()
   LIN {X -3.280, Y -27.534, Z 63.750}
   LaserStart_Ext()
   LIN {X -3.280, Y -25.236, Z 63.750}
   LaserEnd_Ext()
   LIN {X -3.280, Y -15.379, Z 63.750}
   LaserStart_Ext()
   LIN {X -3.280, Y -5.198, Z 63.750}
   LaserEnd_Ext()
   LIN {X -3.280, Y 30.517, Z 63.750}
   LaserStart_Ext()
   LIN {X -3.280, Y 44.018, Z 63.750}
   LaserEnd_Ext()
   LIN {X -2.280, Y 43.741, Z 63.750}
   LaserStart_Ext()
   LIN {X -2.280, Y 25.790, Z 63.750}
   LaserEnd_Ext()
   LIN {X -2.280, Y -0.827, Z 63.750}
   LaserStart_Ext()
   LIN {X -2.280, Y -14.899, Z 63.750}
   LaserEnd_Ext()
   LIN {X -2.280, Y -25.817, Z 63.750}
   LaserStart_Ext()
   LIN {X -2.280, Y -27.769, Z 63.750}
   LaserEnd_Ext()
   LIN {X -1.280, Y -28.004, Z 63.750}
   LaserStart_Ext()
   LIN {X -1.280, Y -26.120, Z 63.750}
   LaserEnd_Ext()
   LIN {X -1.280, Y -14.573, Z 63.750}
   LaserStart_Ext()
   LIN {X -1.280, Y 7.723, Z 63.750}
   LaserEnd_Ext()
   LIN {X -1.280, Y 16.394, Z 63.750}
   LaserStart_Ext()
   LIN {X -1.280, Y 42.958, Z 63.750}
   LaserEnd_Ext()
   LIN {X -0.280, Y 41.135, Z 63.750}
   LaserStart_Ext()
   LIN {X -0.280, Y -14.351, Z 63.750}
   LaserEnd_Ext()
   LIN {X -0.280, Y -26.227, Z 63.750}
   LaserStart_Ext()
   LIN {X -0.280, Y -28.240, Z 63.750}
   LaserEnd_Ext()
   LIN {X 0.720, Y -28.201, Z 63.750}
   LaserStart_Ext()
   LIN {X 0.720, Y -26.274, Z 63.750}
   LaserEnd_Ext()
   LIN {X 0.720, Y -14.457, Z 63.750}
   LaserStart_Ext()
   LIN {X 0.720, Y 38.830, Z 63.750}
   LaserEnd_Ext()
   LIN {X 1.720, Y 36.385, Z 63.750}
   LaserStart_Ext()
   LIN {X 1.720, Y -14.563, Z 63.750}
   LaserEnd_Ext()
   LIN {X 1.720, Y -25.961, Z 63.750}
   LaserStart_Ext()
   LIN {X 1.720, Y -28.029, Z 63.750}
   LaserEnd_Ext()
   LIN {X 2.720, Y -27.822, Z 63.750}
   LaserStart_Ext()
   LIN {X 2.720, Y -25.645, Z 63.750}
   LaserEnd_Ext()
   LIN {X 2.720, Y -15.049, Z 63.750}
   LaserStart_Ext()
   LIN {X 2.720, Y 33.732, Z 63.750}
   LaserEnd_Ext()
   LIN {X 3.720, Y 30.783, Z 63.750}
   LaserStart_Ext()
   LIN {X 3.720, Y -15.637, Z 63.750}
   LaserEnd_Ext()
   LIN {X 3.720, Y -24.916, Z 63.750}
   LaserStart_Ext()
   LIN {X 3.720, Y -27.277, Z 63.750}
   LaserEnd_Ext()
   LIN {X 4.720, Y -26.732, Z 63.750}
   LaserStart_Ext()
   LIN {X 4.720, Y -24.018, Z 63.750}
   LaserEnd_Ext()
   LIN {X 4.720, Y -16.773, Z 63.750}
   LaserStart_Ext()
   LIN {X 4.720, Y 27.661, Z 63.750}
   LaserEnd_Ext()
   LIN {X 5.720, Y 24.024, Z 63.750}
   LaserStart_Ext()
   LIN {X 5.720, Y -18.367, Z 63.750}
   LaserEnd_Ext()
   LIN {X 5.720, Y -21.869, Z 63.750}
   LaserStart_Ext()
   LIN {X 5.720, Y -25.662, Z 63.750}
   LaserEnd_Ext()
   LIN {X 6.720, Y -24.474, Z 63.750}
   LaserStart_Ext()
   LIN {X 6.720, Y 20.109, Z 63.750}
   LaserEnd_Ext()
   LIN {X 7.720, Y 14.280, Z 63.750}
   LaserStart_Ext()
   LIN {X 7.720, Y -22.191, Z 63.750}
   LaserEnd_Ext()
   LIN {X 8.720, Y -15.898, Z 63.750}
   LaserStart_Ext()
   LIN {X 8.720, Y 7.630, Z 63.750}
   LaserEnd_Ext()
   LIN {X -3.247, Y -24.000, Z 64.600}
   LaserStart_Ext()
   LIN {X -3.733, Y -23.335, Z 64.600} C_DIS
   LIN {X -4.472, Y -22.316, Z 64.600} C_DIS
   LIN {X -4.717, Y -21.109, Z 64.600} C_DIS
   LIN {X -4.890, Y -20.271, Z 64.600} C_DIS
   LIN {X -4.196, Y -18.126, Z 64.600} C_DIS
   LIN {X -3.958, Y -17.390, Z 64.600} C_DIS
   LIN {X -2.437, Y -15.978, Z 64.600} C_DIS
   LIN {X -1.894, Y -15.801, Z 64.600} C_DIS
   LIN {X -0.352, Y -15.291, Z 64.600} C_DIS
   LIN {X 1.576, Y -15.489, Z 64.600} C_DIS
   LIN {X 1.680, Y -15.500, Z 64.600} C_DIS
   LIN {X 3.514, Y -16.573, Z 64.600} C_DIS
   LIN {X 4.677, Y -18.392, Z 64.600} C_DIS
   LIN {X 4.885, Y -18.715, Z 64.600} C_DIS
   LIN {X 4.913, Y -19.028, Z 64.600} C_DIS
   LIN {X 5.075, Y -20.917, Z 64.600} C_DIS
   LIN {X 4.588, Y -22.165, Z 64.600} C_DIS
   LIN {X 4.178, Y -23.161, Z 64.600} C_DIS
   LIN {X 2.617, Y -24.571, Z 64.600} C_DIS
   LIN {X 2.428, Y -24.668, Z 64.600} C_DIS
   LIN {X 0.575, Y -25.249, Z 64.600} C_DIS
   LIN {X -0.681, Y -25.120, Z 64.600} C_DIS
   LIN {X -1.460, Y -25.036, Z 64.600} C_DIS
   LIN {X -2.405, Y -24.487, Z 64.600} C_DIS
   LIN {X -3.247, Y -24.000, Z 64.600}
   LaserEnd_Ext()
   LIN {X -5.551, Y 34.792, Z 64.600}
   LaserStart_Ext()
   LIN {X -6.313, Y 37.037, Z 64.600} C_DIS
   LIN {X -6.847, Y 38.481, Z 64.600} C_DIS
   LIN {X -7.317, Y 39.705, Z 64.600} C_DIS
   LIN {X -7.509, Y 40.668, Z 64.600} C_DIS
   LIN {X -7.612, Y 41.128, Z 64.600} C_DIS
   LIN {X -7.418, Y 42.115, Z 64.600} C_DIS
   LIN {X -7.269, Y 42.824, Z 64.600} C_DIS
   LIN {X -7.090, Y 43.084, Z 64.600} C_DIS
   LIN {X -6.267, Y 44.180, Z 64.600} C_DIS
   LIN {X -4.953, Y 44.787, Z 64.600} C_DIS
   LIN {X -4.086, Y 45.150, Z 64.600} C_DIS
   LIN {X -3.061, Y 45.038, Z 64.600} C_DIS
   LIN {X -2.351, Y 44.959, Z 64.600} C_DIS
   LIN {X -1.469, Y 44.419, Z 64.600} C_DIS
   LIN {X -0.866, Y 44.051, Z 64.600} C_DIS
   LIN {X -0.588, Y 43.664, Z 64.600} C_DIS
   LIN {X -0.010, Y 42.854, Z 64.600} C_DIS
   LIN {X 0.501, Y 41.739, Z 64.600} C_DIS
   LIN {X 0.609, Y 41.506, Z 64.600} C_DIS
   LIN {X 0.712, Y 41.272, Z 64.600} C_DIS
   LIN {X 1.437, Y 39.621, Z 64.600} C_DIS
   LIN {X 1.711, Y 38.936, Z 64.600} C_DIS
   LIN {X 2.561, Y 36.898, Z 64.600} C_DIS
   LIN {X 3.847, Y 33.493, Z 64.600} C_DIS
   LIN {X 4.149, Y 32.672, Z 64.600} C_DIS
   LIN {X 4.608, Y 31.222, Z 64.600} C_DIS
   LIN {X 6.034, Y 26.809, Z 64.600} C_DIS
   LIN {X 7.459, Y 21.189, Z 64.600} C_DIS
   LIN {X 7.861, Y 19.619, Z 64.600} C_DIS
   LIN {X 8.143, Y 18.138, Z 64.600} C_DIS
   LIN {X 9.493, Y 9.160, Z 64.600} C_DIS
   LIN {X 9.955, Y 6.191, Z 64.600} C_DIS
   LIN {X 9.979, Y 5.975, Z 64.600} C_DIS
   LIN {X 9.991, Y 5.781, Z 64.600} C_DIS
   LIN {X 10.026, Y 5.221, Z 64.600} C_DIS
   LIN {X 10.372, Y -0.392, Z 64.600} C_DIS
   LIN {X 10.396, Y -4.292, Z 64.600} C_DIS
   LIN {X 10.394, Y -6.906, Z 64.600} C_DIS
   LIN {X 10.177, Y -11.478, Z 64.600} C_DIS
   LIN {X 10.165, Y -11.689, Z 64.600} C_DIS
   LIN {X 10.127, Y -12.119, Z 64.600} C_DIS
   LIN {X 9.836, Y -15.481, Z 64.600} C_DIS
   LIN {X 9.692, Y -16.736, Z 64.600} C_DIS
   LIN {X 9.489, Y -18.421, Z 64.600} C_DIS
   LIN {X 9.035, Y -21.540, Z 64.600} C_DIS
   LIN {X 9.018, Y -21.651, Z 64.600} C_DIS
   LIN {X 8.971, Y -21.788, Z 64.600} C_DIS
   LIN {X 8.075, Y -24.446, Z 64.600} C_DIS
   LIN {X 6.413, Y -26.439, Z 64.600} C_DIS
   LIN {X 5.639, Y -27.356, Z 64.600} C_DIS
   LIN {X 4.451, Y -28.004, Z 64.600} C_DIS
   LIN {X 3.004, Y -28.789, Z 64.600} C_DIS
   LIN {X 1.768, Y -28.992, Z 64.600} C_DIS
   LIN {X 0.070, Y -29.285, Z 64.600} C_DIS
   LIN {X -3.978, Y -28.331, Z 64.600} C_DIS
   LIN {X -4.074, Y -28.263, Z 64.600} C_DIS
   LIN {X -6.330, Y -26.621, Z 64.600} C_DIS
   LIN {X -7.375, Y -24.989, Z 64.600} C_DIS
   LIN {X -8.342, Y -23.457, Z 64.600} C_DIS
   LIN {X -8.654, Y -21.318, Z 64.600} C_DIS
   LIN {X -8.885, Y -19.787, Z 64.600} C_DIS
   LIN {X -8.546, Y -18.368, Z 64.600} C_DIS
   LIN {X -8.142, Y -16.705, Z 64.600} C_DIS
   LIN {X -7.584, Y -15.366, Z 64.600} C_DIS
   LIN {X -7.008, Y -13.965, Z 64.600} C_DIS
   LIN {X -6.150, Y -11.566, Z 64.600} C_DIS
   LIN {X -5.709, Y -10.350, Z 64.600} C_DIS
   LIN {X -5.360, Y -9.201, Z 64.600} C_DIS
   LIN {X -4.602, Y -6.670, Z 64.600} C_DIS
   LIN {X -4.199, Y -4.832, Z 64.600} C_DIS
   LIN {X -3.194, Y -0.439, Z 64.600} C_DIS
   LIN {X -2.486, Y 4.742, Z 64.600} C_DIS
   LIN {X -2.350, Y 5.752, Z 64.600} C_DIS
   LIN {X -2.135, Y 11.349, Z 64.600} C_DIS
   LIN {X -2.106, Y 14.785, Z 64.600} C_DIS
   LIN {X -2.460, Y 18.113, Z 64.600} C_DIS
   LIN {X -2.957, Y 23.946, Z 64.600} C_DIS
   LIN {X -3.404, Y 26.212, Z 64.600} C_DIS
   LIN {X -3.830, Y 28.477, Z 64.600} C_DIS
   LIN {X -4.789, Y 32.262, Z 64.600} C_DIS
   LIN {X -5.551, Y 34.792, Z 64.600}
   LaserEnd_Ext()
   LIN {X -3.615, Y -27.360, Z 64.600}
   LaserStart_Ext()
   LIN {X 3.540, Y -27.360, Z 64.600}
   LaserEnd_Ext()
   LIN {X 5.171, Y -26.360, Z 64.600}
   LaserStart_Ext()
   LIN {X -4.989, Y -26.360, Z 64.600}
   LaserEnd_Ext()
   LIN {X -5.950, Y -25.360, Z 64.600}
   LaserStart_Ext()
   LIN {X -2.893, Y -25.360, Z 64.600}
   LaserEnd_Ext()
   LIN {X 3.234, Y -25.360, Z 64.600}
   LaserStart_Ext()
   LIN {X 6.011, Y -25.360, Z 64.600}
   LaserEnd_Ext()
   LIN {X 6.845, Y -24.360, Z 64.600}
   LaserStart_Ext()
   LIN {X 4.343, Y -24.360, Z 64.600}
   LaserEnd_Ext()
   LIN {X -4.223, Y -24.360, Z 64.600}
   LaserStart_Ext()
   LIN {X -6.589, Y -24.360, Z 64.600}
   LaserEnd_Ext()
   LIN {X -7.220, Y -23.360, Z 64.600}
   LaserStart_Ext()
   LIN {X -4.950, Y -23.360, Z 64.600}
   LaserEnd_Ext()
   LIN {X 5.178, Y -23.360, Z 64.600}
   LaserStart_Ext()
   LIN {X 7.386, Y -23.360, Z 64.600}
   LaserEnd_Ext()
   LIN {X 7.723, Y -22.360, Z 64.600}
   LaserStart_Ext()
   LIN {X 5.586, Y -22.360, Z 64.600}
   LaserEnd_Ext()
   LIN {X -5.483, Y -22.360, Z 64.600}
   LaserStart_Ext()
   LIN {X -7.491, Y -22.360, Z 64.600}
   LaserEnd_Ext()
   LIN {X -7.637, Y -21.360, Z 64.600}
   LaserStart_Ext()
   LIN {X -5.687, Y -21.360, Z 64.600}
   LaserEnd_Ext()
   LIN {X 5.975, Y -21.360, Z 64.600}
   LaserStart_Ext()
   LIN {X 8.051, Y -21.360, Z 64.600}
   LaserEnd_Ext()
   LIN {X 8.196, Y -20.360, Z 64.600}
   LaserStart_Ext()
   LIN {X 6.031, Y -20.360, Z 64.600}
   LaserEnd_Ext()
   LIN {X -5.886, Y -20.360, Z 64.600}
   LaserStart_Ext()
   LIN {X -7.787, Y -20.360, Z 64.600}
   LaserEnd_Ext()
   LIN {X -7.755, Y -19.360, Z 64.600}
   LaserStart_Ext()
   LIN {X -5.646, Y -19.360, Z 64.600}
   LaserEnd_Ext()
   LIN {X 5.945, Y -19.360, Z 64.600}
   LaserStart_Ext()
   LIN {X 8.342, Y -19.360, Z 64.600}
   LaserEnd_Ext()
   LIN {X 8.488, Y -18.360, Z 64.600}
   LaserStart_Ext()
   LIN {X 5.820, Y -18.360, Z 64.600}
   LaserEnd_Ext()
   LIN {X -5.323, Y -18.360, Z 64.600}
   LaserStart_Ext()
   LIN {X -7.515, Y -18.360, Z 64.600}
   LaserEnd_Ext()
   LIN {X -7.272, Y -17.360, Z 64.600}
   LaserStart_Ext()
   LIN {X -4.999, Y -17.360, Z 64.600}
   LaserEnd_Ext()
   LIN {X 5.204, Y -17.360, Z 64.600}
   LaserStart_Ext()
   LIN {X 8.610, Y -17.360, Z 64.600}
   LaserEnd_Ext()
   LIN {X 8.729, Y -16.360, Z 64.600}
   LaserStart_Ext()
   LIN {X 4.565, Y -16.360, Z 64.600}
   LaserEnd_Ext()
   LIN {X -4.319, Y -16.360, Z 64.600}
   LaserStart_Ext()
   LIN {X -6.915, Y -16.360, Z 64.600}
   LaserEnd_Ext()
   LIN {X -6.500, Y -15.360, Z 64.600}
   LaserStart_Ext()
   LIN {X -3.241, Y -15.360, Z 64.600}
   LaserEnd_Ext()
   LIN {X 3.420, Y -15.360, Z 64.600}
   LaserStart_Ext()
   LIN {X 8.843, Y -15.360, Z 64.600}
   LaserEnd_Ext()
   LIN {X 8.929, Y -14.360, Z 64.600}
   LaserStart_Ext()
   LIN {X 0.373, Y -14.360, Z 64.600}
   LaserEnd_Ext()
   LIN {X -0.723, Y -14.360, Z 64.600}
   LaserStart_Ext()
   LIN {X -6.090, Y -14.360, Z 64.600}
   LaserEnd_Ext()
   LIN {X -5.730, Y -13.360, Z 64.600}
   LaserStart_Ext()
   LIN {X 9.016, Y -13.360, Z 64.600}
   LaserEnd_Ext()
   LIN {X 9.102, Y -12.360, Z 64.600}
   LaserStart_Ext()
   LIN {X -5.372, Y -12.360, Z 64.600}
   LaserEnd_Ext()
   LIN {X -5.011, Y -11.360, Z 64.600}
   LaserStart_Ext()
   LIN {X 9.181, Y -11.360, Z 64.600}
   LaserEnd_Ext()
   LIN {X 9.229, Y -10.360, Z 64.600}
   LaserStart_Ext()
   LIN {X -4.667, Y -10.360, Z 64.600}
   LaserEnd_Ext()
   LIN {X -4.363, Y -9.360, Z 64.600}
   LaserStart_Ext()
   LIN {X 9.276, Y -9.360, Z 64.600}
   LaserEnd_Ext()
   LIN {X 9.324, Y -8.360, Z 64.600}
   LaserStart_Ext()
   LIN {X -4.064, Y -8.360, Z 64.600}
   LaserEnd_Ext()
   LIN {X -3.764, Y -7.360, Z 64.600}
   LaserStart_Ext()
   LIN {X 9.371, Y -7.360, Z 64.600}
   LaserEnd_Ext()
   LIN {X 9.394, Y -6.360, Z 64.600}
   LaserStart_Ext()
   LIN {X -3.510, Y -6.360, Z 64.600}
   LaserEnd_Ext()
   LIN {X -3.291, Y -5.360, Z 64.600}
   LaserStart_Ext()
   LIN {X 9.395, Y -5.360, Z 64.600}
   LaserEnd_Ext()
   LIN {X 9.396, Y -4.360, Z 64.600}
   LaserStart_Ext()
   LIN {X -3.065, Y -4.360, Z 64.600}
   LaserEnd_Ext()
   LIN {X -2.837, Y -3.360, Z 64.600}
   LaserStart_Ext()
   LIN {X 9.390, Y -3.360, Z 64.600}
   LaserEnd_Ext()
   LIN {X 9.384, Y -2.360, Z 64.600}
   LaserStart_Ext()
   LIN {X -2.608, Y -2.360, Z 64.600}
   LaserEnd_Ext()
   LIN {X -2.379, Y -1.360, Z 64.600}
   LaserStart_Ext()
   LIN {X 9.378, Y -1.360, Z 64.600}
   LaserEnd_Ext()
   LIN {X 9.368, Y -0.360, Z 64.600}
   LaserStart_Ext()
   LIN {X -2.174, Y -0.360, Z 64.600}
   LaserEnd_Ext()
   LIN {X -2.037, Y 0.640, Z 64.600}
   LaserStart_Ext()
   LIN {X 9.306, Y 0.640, Z 64.600}
   LaserEnd_Ext()
   LIN {X 9.245, Y 1.640, Z 64.600}
   LaserStart_Ext()
   LIN {X -1.901, Y 1.640, Z 64.600}
   LaserEnd_Ext()
   LIN {X -1.764, Y 2.640, Z 64.600}
   LaserStart_Ext()
   LIN {X 9.183, Y 2.640, Z 64.600}
   LaserEnd_Ext()
   LIN {X 9.121, Y 3.640, Z 64.600}
   LaserStart_Ext()
   LIN {X -1.628, Y 3.640, Z 64.600}
   LaserEnd_Ext()
   LIN {X -1.491, Y 4.640, Z 64.600}
   LaserStart_Ext()
   LIN {X 9.060, Y 4.640, Z 64.600}
   LaserEnd_Ext()
   LIN {X 8.998, Y 5.640, Z 64.600}
   LaserStart_Ext()
   LIN {X -1.357, Y 5.640, Z 64.600}
   LaserEnd_Ext()
   LIN {X -1.315, Y 6.640, Z 64.600}
   LaserStart_Ext()
   LIN {X 8.873, Y 6.640, Z 64.600}
   LaserEnd_Ext()
   LIN {X 8.717, Y 7.640, Z 64.600}
   LaserStart_Ext()
   LIN {X -1.277, Y 7.640, Z 64.600}
   LaserEnd_Ext()
   LIN {X -1.238, Y 8.640, Z 64.600}
   LaserStart_Ext()
   LIN {X 8.562, Y 8.640, Z 64.600}
   LaserEnd_Ext()
   LIN {X 8.410, Y 9.640, Z 64.600}
   LaserStart_Ext()
   LIN {X -1.200, Y 9.640, Z 64.600}
   LaserEnd_Ext()
   LIN {X -1.161, Y 10.640, Z 64.600}
   LaserStart_Ext()
   LIN {X 8.259, Y 10.640, Z 64.600}
   LaserEnd_Ext()
   LIN {X 8.109, Y 11.640, Z 64.600}
   LaserStart_Ext()
   LIN {X -1.132, Y 11.640, Z 64.600}
   LaserEnd_Ext()
   LIN {X -1.124, Y 12.640, Z 64.600}
   LaserStart_Ext()
   LIN {X 7.958, Y 12.640, Z 64.600}
   LaserEnd_Ext()
   LIN {X 7.808, Y 13.640, Z 64.600}
   LaserStart_Ext()
   LIN {X -1.116, Y 13.640, Z 64.600}
   LaserEnd_Ext()
   LIN {X -1.108, Y 14.640, Z 64.600}
   LaserStart_Ext()
   LIN {X 7.658, Y 14.640, Z 64.600}
   LaserEnd_Ext()
   LIN {X 7.507, Y 15.640, Z 64.600}
   LaserStart_Ext()
   LIN {X -1.192, Y 15.640, Z 64.600}
   LaserEnd_Ext()
   LIN {X -1.298, Y 16.640, Z 64.600}
   LaserStart_Ext()
   LIN {X 7.357, Y 16.640, Z 64.600}
   LaserEnd_Ext()
   LIN {X 7.207, Y 17.640, Z 64.600}
   LaserStart_Ext()
   LIN {X -1.404, Y 17.640, Z 64.600}
   LaserEnd_Ext()
   LIN {X -1.501, Y 18.640, Z 64.600}
   LaserStart_Ext()
   LIN {X 7.030, Y 18.640, Z 64.600}
   LaserEnd_Ext()
   LIN {X 6.824, Y 19.640, Z 64.600}
   LaserStart_Ext()
   LIN {X -1.586, Y 19.640, Z 64.600}
   LaserEnd_Ext()
   LIN {X -1.672, Y 20.640, Z 64.600}
   LaserStart_Ext()
   LIN {X 6.567, Y 20.640, Z 64.600}
   LaserEnd_Ext()
   LIN {X 6.313, Y 21.640, Z 64.600}
   LaserStart_Ext()
   LIN {X -1.757, Y 21.640, Z 64.600}
   LaserEnd_Ext()
   LIN {X -1.842, Y 22.640, Z 64.600}
   LaserStart_Ext()
   LIN {X 6.059, Y 22.640, Z 64.600}
   LaserEnd_Ext()
   LIN {X 5.806, Y 23.640, Z 64.600}
   LaserStart_Ext()
   LIN {X -1.927, Y 23.640, Z 64.600}
   LaserEnd_Ext()
   LIN {X -2.075, Y 24.640, Z 64.600}
   LaserStart_Ext()
   LIN {X 5.552, Y 24.640, Z 64.600}
   LaserEnd_Ext()
   LIN {X 5.299, Y 25.640, Z 64.600}
   LaserStart_Ext()
   LIN {X -2.272, Y 25.640, Z 64.600}
   LaserEnd_Ext()
   LIN {X -2.467, Y 26.640, Z 64.600}
   LaserStart_Ext()
   LIN {X 5.037, Y 26.640, Z 64.600}
   LaserEnd_Ext()
   LIN {X 4.714, Y 27.640, Z 64.600}
   LaserStart_Ext()
   LIN {X -2.655, Y 27.640, Z 64.600}
   LaserEnd_Ext()
   LIN {X -2.843, Y 28.640, Z 64.600}
   LaserStart_Ext()
   LIN {X 4.391, Y 28.640, Z 64.600}
   LaserEnd_Ext()
   LIN {X 4.068, Y 29.640, Z 64.600}
   LaserStart_Ext()
   LIN {X -3.093, Y 29.640, Z 64.600}
   LaserEnd_Ext()
   LIN {X -3.346, Y 30.640, Z 64.600}
   LaserStart_Ext()
   LIN {X 3.745, Y 30.640, Z 64.600}
   LaserEnd_Ext()
   LIN {X 3.427, Y 31.640, Z 64.600}
   LaserStart_Ext()
   LIN {X -3.600, Y 31.640, Z 64.600}
   LaserEnd_Ext()
   LIN {X -3.858, Y 32.640, Z 64.600}
   LaserStart_Ext()
   LIN {X 3.096, Y 32.640, Z 64.600}
   LaserEnd_Ext()
   LIN {X 2.723, Y 33.640, Z 64.600}
   LaserStart_Ext()
   LIN {X -4.159, Y 33.640, Z 64.600}
   LaserEnd_Ext()
   LIN {X -4.461, Y 34.640, Z 64.600}
   LaserStart_Ext()
   LIN {X 2.345, Y 34.640, Z 64.600}
   LaserEnd_Ext()
   LIN {X 1.967, Y 35.640, Z 64.600}
   LaserStart_Ext()
   LIN {X -4.783, Y 35.640, Z 64.600}
   LaserEnd_Ext()
   LIN {X -5.122, Y 36.640, Z 64.600}
   LaserStart_Ext()
   LIN {X 1.585, Y 36.640, Z 64.600}
   LaserEnd_Ext()
   LIN {X 1.168, Y 37.640, Z 64.600}
   LaserStart_Ext()
   LIN {X -5.470, Y 37.640, Z 64.600}
   LaserEnd_Ext()
   LIN {X -5.840, Y 38.640, Z 64.600}
   LaserStart_Ext()
   LIN {X 0.753, Y 38.640, Z 64.600}
   LaserEnd_Ext()
   LIN {X 0.337, Y 39.640, Z 64.600}
   LaserStart_Ext()
   LIN {X -6.221, Y 39.640, Z 64.600}
   LaserEnd_Ext()
   LIN {X -6.484, Y 40.640, Z 64.600}
   LaserStart_Ext()
   LIN {X -0.102, Y 40.640, Z 64.600}
   LaserEnd_Ext()
   LIN {X -0.554, Y 41.640, Z 64.600}
   LaserStart_Ext()
   LIN {X -6.492, Y 41.640, Z 64.600}
   LaserEnd_Ext()
   LIN {X -6.173, Y 42.640, Z 64.600}
   LaserStart_Ext()
   LIN {X -1.086, Y 42.640, Z 64.600}
   LaserEnd_Ext()
   LIN {X -2.112, Y 43.640, Z 64.600}
   LaserStart_Ext()
   LIN {X -5.052, Y 43.640, Z 64.600}
   LaserEnd_Ext()
   LIN {X 5.120, Y -20.443, Z 65.450}
   LaserStart_Ext()
   LIN {X 5.155, Y -20.852, Z 65.450} C_DIS
   LIN {X 4.356, Y -22.903, Z 65.450} C_DIS
   LIN {X 4.291, Y -23.061, Z 65.450} C_DIS
   LIN {X 4.017, Y -23.308, Z 65.450} C_DIS
   LIN {X 2.676, Y -24.549, Z 65.450} C_DIS
   LIN {X 1.547, Y -24.919, Z 65.450} C_DIS
   LIN {X 0.666, Y -25.195, Z 65.450} C_DIS
   LIN {X -0.701, Y -25.054, Z 65.450} C_DIS
   LIN {X -1.370, Y -24.987, Z 65.450} C_DIS
   LIN {X -1.805, Y -24.738, Z 65.450} C_DIS
   LIN {X -3.160, Y -23.955, Z 65.450} C_DIS
   LIN {X -4.254, Y -22.457, Z 65.450} C_DIS
   LIN {X -4.389, Y -22.274, Z 65.450} C_DIS
   LIN {X -4.437, Y -22.045, Z 65.450} C_DIS
   LIN {X -4.812, Y -20.230, Z 65.450} C_DIS
   LIN {X -4.446, Y -19.100, Z 65.450} C_DIS
   LIN {X -3.874, Y -17.330, Z 65.450} C_DIS
   LIN {X -2.888, Y -16.414, Z 65.450} C_DIS
   LIN {X -2.358, Y -15.925, Z 65.450} C_DIS
   LIN {X -0.285, Y -15.239, Z 65.450} C_DIS
   LIN {X 0.497, Y -15.320, Z 65.450} C_DIS
   LIN {X 1.747, Y -15.444, Z 65.450} C_DIS
   LIN {X 3.270, Y -16.329, Z 65.450} C_DIS
   LIN {X 3.584, Y -16.512, Z 65.450} C_DIS
   LIN {X 3.772, Y -16.807, Z 65.450} C_DIS
   LIN {X 4.960, Y -18.650, Z 65.450} C_DIS
   LIN {X 5.120, Y -20.443, Z 65.450}
   LaserEnd_Ext()
   LIN {X -8.256, Y -23.425, Z 65.450}
   LaserStart_Ext()
   LIN {X -8.321, Y -22.977, Z 65.450} C_DIS
   LIN {X -8.807, Y -19.755, Z 65.450} C_DIS
   LIN {X -8.096, Y -16.771, Z 65.450} C_DIS
   LIN {X -8.071, Y -16.671, Z 65.450} C_DIS
   LIN {X -6.944, Y -13.927, Z 65.450} C_DIS
   LIN {X -5.898, Y -11.007, Z 65.450} C_DIS
   LIN {X -5.653, Y -10.308, Z 65.450} C_DIS
   LIN {X -5.431, Y -9.553, Z 65.450} C_DIS
   LIN {X -4.554, Y -6.624, Z 65.450} C_DIS
   LIN {X -3.827, Y -3.306, Z 65.450} C_DIS
   LIN {X -3.167, Y -0.420, Z 65.450} C_DIS
   LIN {X -2.702, Y 2.984, Z 65.450} C_DIS
   LIN {X -2.350, Y 5.590, Z 65.450} C_DIS
   LIN {X -2.157, Y 10.590, Z 65.450} C_DIS
   LIN {X -2.121, Y 15.001, Z 65.450} C_DIS
   LIN {X -2.575, Y 19.273, Z 65.450} C_DIS
   LIN {X -2.972, Y 23.930, Z 65.450} C_DIS
   LIN {X -3.622, Y 27.221, Z 65.450} C_DIS
   LIN {X -3.866, Y 28.523, Z 65.450} C_DIS
   LIN {X -4.418, Y 30.701, Z 65.450} C_DIS
   LIN {X -4.819, Y 32.255, Z 65.450} C_DIS
   LIN {X -5.062, Y 33.042, Z 65.450} C_DIS
   LIN {X -5.602, Y 34.831, Z 65.450} C_DIS
   LIN {X -6.280, Y 36.818, Z 65.450} C_DIS
   LIN {X -6.368, Y 37.074, Z 65.450} C_DIS
   LIN {X -6.429, Y 37.236, Z 65.450} C_DIS
   LIN {X -6.927, Y 38.574, Z 65.450} C_DIS
   LIN {X -7.264, Y 39.444, Z 65.450} C_DIS
   LIN {X -7.379, Y 39.740, Z 65.450} C_DIS
   LIN {X -7.474, Y 40.134, Z 65.450} C_DIS
   LIN {X -7.672, Y 41.018, Z 65.450} C_DIS
   LIN {X -7.527, Y 41.754, Z 65.450} C_DIS
   LIN {X -7.369, Y 42.783, Z 65.450} C_DIS
   LIN {X -6.246, Y 44.286, Z 65.450} C_DIS
   LIN {X -4.160, Y 45.193, Z 65.450} C_DIS
   LIN {X -4.031, Y 45.179, Z 65.450} C_DIS
   LIN {X -2.425, Y 45.005, Z 65.450} C_DIS
   LIN {X -1.832, Y 44.646, Z 65.450} C_DIS
   LIN {X -0.938, Y 44.102, Z 65.450} C_DIS
   LIN {X -0.305, Y 43.220, Z 65.450} C_DIS
   LIN {X -0.080, Y 42.907, Z 65.450} C_DIS
   LIN {X 0.055, Y 42.617, Z 65.450} C_DIS
   LIN {X 0.542, Y 41.559, Z 65.450} C_DIS
   LIN {X 1.312, Y 39.824, Z 65.450} C_DIS
   LIN {X 2.456, Y 37.080, Z 65.450} C_DIS
   LIN {X 4.077, Y 32.789, Z 65.450} C_DIS
   LIN {X 4.141, Y 32.623, Z 65.450} C_DIS
   LIN {X 4.175, Y 32.523, Z 65.450} C_DIS
   LIN {X 6.024, Y 26.800, Z 65.450} C_DIS
   LIN {X 7.922, Y 19.319, Z 65.450} C_DIS
   LIN {X 7.985, Y 19.071, Z 65.450} C_DIS
   LIN {X 8.029, Y 18.838, Z 65.450} C_DIS
   LIN {X 8.242, Y 17.423, Z 65.450} C_DIS
   LIN {X 9.944, Y 6.486, Z 65.450} C_DIS
   LIN {X 10.034, Y 5.691, Z 65.450} C_DIS
   LIN {X 10.046, Y 5.486, Z 65.450} C_DIS
   LIN {X 10.078, Y 4.974, Z 65.450} C_DIS
   LIN {X 10.205, Y 2.912, Z 65.450} C_DIS
   LIN {X 10.404, Y -0.315, Z 65.450} C_DIS
   LIN {X 10.442, Y -6.444, Z 65.450} C_DIS
   LIN {X 10.441, Y -6.829, Z 65.450} C_DIS
   LIN {X 10.404, Y -7.621, Z 65.450} C_DIS
   LIN {X 10.224, Y -11.612, Z 65.450} C_DIS
   LIN {X 10.135, Y -12.729, Z 65.450} C_DIS
   LIN {X 9.904, Y -15.405, Z 65.450} C_DIS
   LIN {X 9.617, Y -17.904, Z 65.450} C_DIS
   LIN {X 9.564, Y -18.346, Z 65.450} C_DIS
   LIN {X 9.431, Y -19.255, Z 65.450} C_DIS
   LIN {X 9.100, Y -21.577, Z 65.450} C_DIS
   LIN {X 8.737, Y -22.672, Z 65.450} C_DIS
   LIN {X 8.162, Y -24.379, Z 65.450} C_DIS
   LIN {X 6.005, Y -26.965, Z 65.450} C_DIS
   LIN {X 5.750, Y -27.278, Z 65.450} C_DIS
   LIN {X 5.528, Y -27.402, Z 65.450} C_DIS
   LIN {X 3.046, Y -28.749, Z 65.450} C_DIS
   LIN {X 0.529, Y -29.162, Z 65.450} C_DIS
   LIN {X 0.122, Y -29.232, Z 65.450} C_DIS
   LIN {X -3.881, Y -28.288, Z 65.450} C_DIS
   LIN {X -4.831, Y -27.606, Z 65.450} C_DIS
   LIN {X -6.236, Y -26.584, Z 65.450} C_DIS
   LIN {X -8.053, Y -23.745, Z 65.450} C_DIS
   LIN {X -8.256, Y -23.425, Z 65.450}
   LaserEnd_Ext()
   LIN {X 8.602, Y 8.606, Z 65.450}
   LaserStart_Ext()
   LIN {X 8.602, Y -17.969, Z 65.450}
   LaserEnd_Ext()
   LIN {X 7.602, Y -22.910, Z 65.450}
   LaserStart_Ext()
   LIN {X 7.602, Y 15.033, Z 65.450}
   LaserEnd_Ext()
   LIN {X 6.602, Y 20.454, Z 65.450}
   LaserStart_Ext()
   LIN {X 6.602, Y -24.688, Z 65.450}
   LaserEnd_Ext()
   LIN {X 5.602, Y -25.887, Z 65.450}
   LaserStart_Ext()
   LIN {X 5.602, Y -22.460, Z 65.450}
   LaserEnd_Ext()
   LIN {X 5.602, Y -17.800, Z 65.450}
   LaserStart_Ext()
   LIN {X 5.602, Y 24.397, Z 65.450}
   LaserEnd_Ext()
   LIN {X 4.602, Y 27.950, Z 65.450}
   LaserStart_Ext()
   LIN {X 4.602, Y -16.248, Z 65.450}
   LaserEnd_Ext()
   LIN {X 4.602, Y -24.130, Z 65.450}
   LaserStart_Ext()
   LIN {X 4.602, Y -26.766, Z 65.450}
   LaserEnd_Ext()
   LIN {X 3.602, Y -27.309, Z 65.450}
   LaserStart_Ext()
   LIN {X 3.602, Y -25.055, Z 65.450}
   LaserEnd_Ext()
   LIN {X 3.602, Y -15.365, Z 65.450}
   LaserStart_Ext()
   LIN {X 3.602, Y 31.045, Z 65.450}
   LaserEnd_Ext()
   LIN {X 2.602, Y 33.865, Z 65.450}
   LaserStart_Ext()
   LIN {X 2.602, Y -14.784, Z 65.450}
   LaserEnd_Ext()
   LIN {X 2.602, Y -25.625, Z 65.450}
   LaserStart_Ext()
   LIN {X 2.602, Y -27.808, Z 65.450}
   LaserEnd_Ext()
   LIN {X 1.602, Y -27.972, Z 65.450}
   LaserStart_Ext()
   LIN {X 1.602, Y -25.950, Z 65.450}
   LaserEnd_Ext()
   LIN {X 1.602, Y -14.424, Z 65.450}
   LaserStart_Ext()
   LIN {X 1.602, Y 36.513, Z 65.450}
   LaserEnd_Ext()
   LIN {X 0.602, Y 38.930, Z 65.450}
   LaserStart_Ext()
   LIN {X 0.602, Y -14.325, Z 65.450}
   LaserEnd_Ext()
   LIN {X 0.602, Y -26.192, Z 65.450}
   LaserStart_Ext()
   LIN {X 0.602, Y -28.137, Z 65.450}
   LaserEnd_Ext()
   LIN {X -0.398, Y -28.082, Z 65.450}
   LaserStart_Ext()
   LIN {X -0.398, Y -26.091, Z 65.450}
   LaserEnd_Ext()
   LIN {X -0.398, Y -14.246, Z 65.450}
   LaserStart_Ext()
   LIN {X -0.398, Y 41.211, Z 65.450}
   LaserEnd_Ext()
   LIN {X -1.398, Y 43.027, Z 65.450}
   LaserStart_Ext()
   LIN {X -1.398, Y 17.660, Z 65.450}
   LaserEnd_Ext()
   LIN {X -1.398, Y 5.166, Z 65.450}
   LaserStart_Ext()
   LIN {X -1.398, Y -14.554, Z 65.450}
   LaserEnd_Ext()
   LIN {X -1.398, Y -25.989, Z 65.450}
   LaserStart_Ext()
   LIN {X -1.398, Y -27.846, Z 65.450}
   LaserEnd_Ext()
   LIN {X -2.398, Y -27.610, Z 65.450}
   LaserStart_Ext()
   LIN {X -2.398, Y -25.550, Z 65.450}
   LaserEnd_Ext()
   LIN {X -2.398, Y -14.885, Z 65.450}
   LaserStart_Ext()
   LIN {X -2.398, Y -1.544, Z 65.450}
   LaserEnd_Ext()
   LIN {X -2.398, Y 26.187, Z 65.450}
   LaserStart_Ext()
   LIN {X -2.398, Y 43.820, Z 65.450}
   LaserEnd_Ext()
   LIN {X -3.398, Y 44.104, Z 65.450}
   LaserStart_Ext()
   LIN {X -3.398, Y 30.747, Z 65.450}
   LaserEnd_Ext()
   LIN {X -3.398, Y -6.021, Z 65.450}
   LaserStart_Ext()
   LIN {X -3.398, Y -15.524, Z 65.450}
   LaserEnd_Ext()
   LIN {X -3.398, Y -24.973, Z 65.450}
   LaserStart_Ext()
   LIN {X -3.398, Y -27.374, Z 65.450}
   LaserEnd_Ext()
   LIN {X -4.398, Y -26.684, Z 65.450}
   LaserStart_Ext()
   LIN {X -4.398, Y -23.955, Z 65.450}
   LaserEnd_Ext()
   LIN {X -4.398, Y -16.451, Z 65.450}
   LaserStart_Ext()
   LIN {X -4.398, Y -9.590, Z 65.450}
   LaserEnd_Ext()
   LIN {X -4.398, Y 34.303, Z 65.450}
   LaserStart_Ext()
   LIN {X -4.398, Y 44.009, Z 65.450}
   LaserEnd_Ext()
   LIN {X -5.398, Y 43.591, Z 65.450}
   LaserStart_Ext()
   LIN {X -5.398, Y 37.327, Z 65.450}
   LaserEnd_Ext()
   LIN {X -5.398, Y -12.576, Z 65.450}
   LaserStart_Ext()
   LIN {X -5.398, Y -18.795, Z 65.450}
   LaserEnd_Ext()
   LIN {X -5.398, Y -22.333, Z 65.450}
   LaserStart_Ext()
   LIN {X -5.398, Y -25.957, Z 65.450}
   LaserEnd_Ext()
   LIN {X -6.398, Y -24.476, Z 65.450}
   LaserStart_Ext()
   LIN {X -6.398, Y -15.230, Z 65.450}
   LaserEnd_Ext()
   LIN {X -6.398, Y 39.977, Z 65.450}
   LaserStart_Ext()
   LIN {X -6.398, Y 42.412, Z 65.450}
   LaserEnd_Ext()
   LIN {X -7.398, Y -18.157, Z 65.450}
   LaserStart_Ext()
   LIN {X -7.398, Y -22.390, Z 65.450}
   LaserEnd_Ext()
   LIN {X 3.598, Y -23.733, Z 66.300}
   LaserStart_Ext()
   LIN {X 2.805, Y -24.466, Z 66.300} C_DIS
   LIN {X 1.255, Y -24.974, Z 66.300} C_DIS
   LIN {X 0.756, Y -25.141, Z 66.300} C_DIS
   LIN {X 0.439, Y -25.111, Z 66.300} C_DIS
   LIN {X -1.280, Y -24.938, Z 66.300} C_DIS
   LIN {X -2.899, Y -24.011, Z 66.300} C_DIS
   LIN {X -3.072, Y -23.910, Z 66.300} C_DIS
   LIN {X -3.213, Y -23.718, Z 66.300} C_DIS
   LIN {X -4.305, Y -22.231, Z 66.300} C_DIS
   LIN {X -4.694, Y -20.375, Z 66.300} C_DIS
   LIN {X -4.733, Y -20.189, Z 66.300} C_DIS
   LIN {X -4.695, Y -20.073, Z 66.300} C_DIS
   LIN {X -3.790, Y -17.269, Z 66.300} C_DIS
   LIN {X -3.711, Y -17.196, Z 66.300} C_DIS
   LIN {X -2.271, Y -15.867, Z 66.300} C_DIS
   LIN {X -0.218, Y -15.187, Z 66.300} C_DIS
   LIN {X 0.493, Y -15.256, Z 66.300} C_DIS
   LIN {X 1.815, Y -15.387, Z 66.300} C_DIS
   LIN {X 2.713, Y -15.909, Z 66.300} C_DIS
   LIN {X 3.654, Y -16.451, Z 66.300} C_DIS
   LIN {X 4.436, Y -17.656, Z 66.300} C_DIS
   LIN {X 5.036, Y -18.586, Z 66.300} C_DIS
   LIN {X 5.126, Y -19.604, Z 66.300} C_DIS
   LIN {X 5.235, Y -20.787, Z 66.300} C_DIS
   LIN {X 4.995, Y -21.411, Z 66.300} C_DIS
   LIN {X 4.379, Y -22.996, Z 66.300} C_DIS
   LIN {X 3.598, Y -23.733, Z 66.300}
   LaserEnd_Ext()
   LIN {X 7.977, Y 19.103, Z 66.300}
   LaserStart_Ext()
   LIN {X 7.626, Y 20.438, Z 66.300} C_DIS
   LIN {X 6.015, Y 26.791, Z 66.300} C_DIS
   LIN {X 4.577, Y 31.241, Z 66.300} C_DIS
   LIN {X 4.216, Y 32.350, Z 66.300} C_DIS
   LIN {X 3.928, Y 33.142, Z 66.300} C_DIS
   LIN {X 2.709, Y 36.318, Z 66.300} C_DIS
   LIN {X 2.352, Y 37.263, Z 66.300} C_DIS
   LIN {X 2.099, Y 37.868, Z 66.300} C_DIS
   LIN {X 1.258, Y 39.862, Z 66.300} C_DIS
   LIN {X 0.518, Y 41.520, Z 66.300} C_DIS
   LIN {X 0.476, Y 41.613, Z 66.300} C_DIS
   LIN {X 0.432, Y 41.708, Z 66.300} C_DIS
   LIN {X -0.149, Y 42.959, Z 66.300} C_DIS
   LIN {X -0.791, Y 43.850, Z 66.300} C_DIS
   LIN {X -1.010, Y 44.152, Z 66.300} C_DIS
   LIN {X -1.712, Y 44.575, Z 66.300} C_DIS
   LIN {X -2.499, Y 45.052, Z 66.300} C_DIS
   LIN {X -2.925, Y 45.098, Z 66.300} C_DIS
   LIN {X -4.235, Y 45.235, Z 66.300} C_DIS
   LIN {X -5.298, Y 44.790, Z 66.300} C_DIS
   LIN {X -6.384, Y 44.281, Z 66.300} C_DIS
   LIN {X -7.275, Y 42.976, Z 66.300} C_DIS
   LIN {X -7.492, Y 42.686, Z 66.300} C_DIS
   LIN {X -7.575, Y 42.147, Z 66.300} C_DIS
   LIN {X -7.734, Y 40.982, Z 66.300} C_DIS
   LIN {X -7.574, Y 40.326, Z 66.300} C_DIS
   LIN {X -7.441, Y 39.775, Z 66.300} C_DIS
   LIN {X -7.175, Y 39.093, Z 66.300} C_DIS
   LIN {X -6.986, Y 38.609, Z 66.300} C_DIS
   LIN {X -6.792, Y 38.094, Z 66.300} C_DIS
   LIN {X -6.424, Y 37.111, Z 66.300} C_DIS
   LIN {X -5.943, Y 35.712, Z 66.300} C_DIS
   LIN {X -5.652, Y 34.870, Z 66.300} C_DIS
   LIN {X -5.332, Y 33.810, Z 66.300} C_DIS
   LIN {X -4.847, Y 32.240, Z 66.300} C_DIS
   LIN {X -4.047, Y 29.140, Z 66.300} C_DIS
   LIN {X -3.903, Y 28.570, Z 66.300} C_DIS
   LIN {X -3.839, Y 28.230, Z 66.300} C_DIS
   LIN {X -2.987, Y 23.914, Z 66.300} C_DIS
   LIN {X -2.690, Y 20.433, Z 66.300} C_DIS
   LIN {X -2.136, Y 15.217, Z 66.300} C_DIS
   LIN {X -2.180, Y 9.832, Z 66.300} C_DIS
   LIN {X -2.350, Y 5.429, Z 66.300} C_DIS
   LIN {X -2.917, Y 1.226, Z 66.300} C_DIS
   LIN {X -3.139, Y -0.400, Z 66.300} C_DIS
   LIN {X -3.455, Y -1.779, Z 66.300} C_DIS
   LIN {X -4.506, Y -6.579, Z 66.300} C_DIS
   LIN {X -4.866, Y -7.782, Z 66.300} C_DIS
   LIN {X -5.597, Y -10.268, Z 66.300} C_DIS
   LIN {X -6.406, Y -12.566, Z 66.300} C_DIS
   LIN {X -6.880, Y -13.890, Z 66.300} C_DIS
   LIN {X -7.409, Y -15.179, Z 66.300} C_DIS
   LIN {X -8.001, Y -16.638, Z 66.300} C_DIS
   LIN {X -8.332, Y -18.054, Z 66.300} C_DIS
   LIN {X -8.730, Y -19.724, Z 66.300} C_DIS
   LIN {X -8.397, Y -21.927, Z 66.300} C_DIS
   LIN {X -8.169, Y -23.392, Z 66.300} C_DIS
   LIN {X -7.093, Y -25.061, Z 66.300} C_DIS
   LIN {X -6.142, Y -26.546, Z 66.300} C_DIS
   LIN {X -5.587, Y -26.950, Z 66.300} C_DIS
   LIN {X -3.783, Y -28.244, Z 66.300} C_DIS
   LIN {X -0.529, Y -29.012, Z 66.300} C_DIS
   LIN {X 0.114, Y -29.176, Z 66.300} C_DIS
   LIN {X 1.211, Y -29.016, Z 66.300} C_DIS
   LIN {X 3.089, Y -28.708, Z 66.300} C_DIS
   LIN {X 4.458, Y -27.965, Z 66.300} C_DIS
   LIN {X 5.924, Y -27.145, Z 66.300} C_DIS
   LIN {X 7.608, Y -25.079, Z 66.300} C_DIS
   LIN {X 8.249, Y -24.311, Z 66.300} C_DIS
   LIN {X 8.420, Y -23.804, Z 66.300} C_DIS
   LIN {X 9.183, Y -21.502, Z 66.300} C_DIS
   LIN {X 9.533, Y -19.045, Z 66.300} C_DIS
   LIN {X 9.638, Y -18.271, Z 66.300} C_DIS
   LIN {X 9.759, Y -17.177, Z 66.300} C_DIS
   LIN {X 9.971, Y -15.328, Z 66.300} C_DIS
   LIN {X 10.092, Y -13.934, Z 66.300} C_DIS
   LIN {X 10.283, Y -11.535, Z 66.300} C_DIS
   LIN {X 10.437, Y -8.110, Z 66.300} C_DIS
   LIN {X 10.489, Y -6.752, Z 66.300} C_DIS
   LIN {X 10.448, Y -2.183, Z 66.300} C_DIS
   LIN {X 10.436, Y -0.238, Z 66.300} C_DIS
   LIN {X 10.384, Y 0.602, Z 66.300} C_DIS
   LIN {X 10.164, Y 4.168, Z 66.300} C_DIS
   LIN {X 10.110, Y 5.053, Z 66.300} C_DIS
   LIN {X 10.088, Y 5.406, Z 66.300} C_DIS
   LIN {X 9.933, Y 6.780, Z 66.300} C_DIS
   LIN {X 8.174, Y 18.084, Z 66.300} C_DIS
   LIN {X 7.977, Y 19.103, Z 66.300}
   LaserEnd_Ext()
   LIN {X -5.648, Y 43.522, Z 66.300}
   LaserStart_Ext()
   LIN {X -1.902, Y 43.522, Z 66.300}
   LaserEnd_Ext()
   LIN {X -1.066, Y 42.522, Z 66.300}
   LaserStart_Ext()
   LIN {X -6.375, Y 42.522, Z 66.300}
   LaserEnd_Ext()
